LIN {X 0,Y 566.195,Z 59.453,A -85,B 0,C 180,E1 -2656.049,E2 -2656.049} C_VEL
LIN {X 0,Y 566.205,Z 59.459,A -85,B 0,C 180,E1 -2659.214,E2 -2659.214} C_VEL
LIN {X 0,Y 566.19,Z 59.456,A -85,B 0,C 180,E1 -2661.637,E2 -2661.637} C_VEL
LIN {X 0,Y 566.175,Z 59.454,A -85,B 0,C 180,E1 -2664.308,E2 -2664.308} C_VEL
LIN {X 0,Y 566.22,Z 59.453,A -85,B 0,C 180,E1 -2666.897,E2 -2666.897} C_VEL
LIN {X 0,Y 566.182,Z 59.457,A -85,B 0,C 180,E1 -2669.407,E2 -2669.407} C_VEL
LIN {X 0,Y 566.213,Z 59.448,A -85,B 0,C 180,E1 -2671.857,E2 -2671.857} C_VEL
LIN {X 0,Y 566.214,Z 59.449,A -85,B 0,C 180,E1 -2674.251,E2 -2674.251} C_VEL
LIN {X 0,Y 566.192,Z 59.462,A -85,B 0,C 180,E1 -2676.714,E2 -2676.714} C_VEL
LIN {X 0,Y 566.214,Z 59.447,A -85,B 0,C 180,E1 -2679.663,E2 -2679.663} C_VEL
LIN {X 0,Y 566.201,Z 59.457,A -85,B 0,C 180,E1 -2682.668,E2 -2682.668} C_VEL
LIN {X 0,Y 566.235,Z 59.447,A -85,B 0,C 180,E1 -2685.626,E2 -2685.626} C_VEL
LIN {X 0,Y 566.235,Z 59.447,A -85,B 0,C 180,E1 -2688.675,E2 -2688.675} C_VEL
LIN {X 0,Y 566.229,Z 59.444,A -85,B 0,C 180,E1 -2691.434,E2 -2691.434} C_VEL
LIN {X 0,Y 566.259,Z 59.451,A -85,B 0,C 180,E1 -2694.301,E2 -2694.301} C_VEL
LIN {X 0,Y 566.284,Z 59.447,A -85,B 0,C 180,E1 -2697.866,E2 -2697.866} C_VEL
LIN {X 0,Y 566.301,Z 59.435,A -85,B 0,C 180,E1 -2700.711,E2 -2700.711} C_VEL
LIN {X 0,Y 566.27,Z 59.442,A -85,B 0,C 180,E1 -2702.845,E2 -2702.845} C_VEL
LIN {X 0,Y 566.258,Z 59.453,A -85,B 0,C 180,E1 -2705.698,E2 -2705.698} C_VEL
LIN {X 0,Y 566.228,Z 59.445,A -85,B 0,C 180,E1 -2708.565,E2 -2708.565} C_VEL
LIN {X 0,Y 566.241,Z 59.45,A -85,B 0,C 180,E1 -2711.454,E2 -2711.454} C_VEL
LIN {X 0,Y 566.233,Z 59.447,A -85,B 0,C 180,E1 -2714.506,E2 -2714.506} C_VEL
LIN {X 0,Y 566.199,Z 59.459,A -85,B 0,C 180,E1 -2717.331,E2 -2717.331} C_VEL
LIN {X 0,Y 566.212,Z 59.447,A -85,B 0,C 180,E1 -2720.337,E2 -2720.337} C_VEL
LIN {X 0,Y 566.188,Z 59.459,A -85,B 0,C 180,E1 -2723.403,E2 -2723.403} C_VEL
LIN {X 0,Y 566.212,Z 59.449,A -85,B 0,C 180,E1 -2725.749,E2 -2725.749} C_VEL
LIN {X 0,Y 566.205,Z 59.452,A -85,B 0,C 180,E1 -2727.48,E2 -2727.48} C_VEL
LIN {X 0,Y 565.532,Z 59.535,A -85,B 0,C 180,E1 -2728.074,E2 -2728.074} C_VEL
LIN {X 0,Y 562.666,Z 59.9,A -85,B 0,C 180,E1 -2729.037,E2 -2729.037} C_VEL
LIN {X 0,Y 560.251,Z 60.196,A -85,B 0,C 180,E1 -2729.813,E2 -2729.813} C_VEL
LIN {X 0,Y 559.223,Z 60.323,A -85,B 0,C 180,E1 -2730.411,E2 -2730.411} C_VEL
LIN {X 0,Y 559.143,Z 60.333,A -85,B 0,C 180,E1 -2730.614,E2 -2730.614} C_VEL
LIN {X 0,Y 559.163,Z 60.326,A -85,B 0,C 180,E1 -2733.574,E2 -2733.574} C_VEL
LIN {X 0,Y 559.167,Z 60.331,A -85,B 0,C 180,E1 -2736.448,E2 -2736.448} C_VEL
LIN {X 0,Y 559.175,Z 60.331,A -85,B 0,C 180,E1 -2738.933,E2 -2738.933} C_VEL
LIN {X 0,Y 559.184,Z 60.325,A -85,B 0,C 180,E1 -2741.768,E2 -2741.768} C_VEL
LIN {X 0,Y 559.136,Z 60.335,A -85,B 0,C 180,E1 -2744.739,E2 -2744.739} C_VEL
LIN {X 0,Y 559.158,Z 60.322,A -85,B 0,C 180,E1 -2747.256,E2 -2747.256} C_VEL
LIN {X 0,Y 559.182,Z 60.329,A -85,B 0,C 180,E1 -2750.135,E2 -2750.135} C_VEL
LIN {X 0,Y 559.144,Z 60.331,A -85,B 0,C 180,E1 -2752.892,E2 -2752.892} C_VEL
LIN {X 0,Y 559.154,Z 60.326,A -85,B 0,C 180,E1 -2755.556,E2 -2755.556} C_VEL
LIN {X 0,Y 559.167,Z 60.336,A -85,B 0,C 180,E1 -2758.137,E2 -2758.137} C_VEL
LIN {X 0,Y 559.14,Z 60.329,A -85,B 0,C 180,E1 -2760.646,E2 -2760.646} C_VEL
LIN {X 0,Y 559.168,Z 60.329,A -85,B 0,C 180,E1 -2763.172,E2 -2763.172} C_VEL
LIN {X 0,Y 559.154,Z 60.335,A -85,B 0,C 180,E1 -2765.495,E2 -2765.495} C_VEL
LIN {X 0,Y 559.169,Z 60.328,A -85,B 0,C 180,E1 -2768.624,E2 -2768.624} C_VEL
LIN {X 0,Y 559.166,Z 60.33,A -85,B 0,C 180,E1 -2770.926,E2 -2770.926} C_VEL
LIN {X 0,Y 559.165,Z 60.332,A -85,B 0,C 180,E1 -2773.948,E2 -2773.948} C_VEL
LIN {X 0,Y 559.17,Z 60.329,A -85,B 0,C 180,E1 -2776.184,E2 -2776.184} C_VEL
LIN {X 0,Y 559.193,Z 60.332,A -85,B 0,C 180,E1 -2779.134,E2 -2779.134} C_VEL
LIN {X 0,Y 559.203,Z 60.325,A -85,B 0,C 180,E1 -2782.054,E2 -2782.054} C_VEL
LIN {X 0,Y 559.253,Z 60.324,A -85,B 0,C 180,E1 -2784.953,E2 -2784.953} C_VEL
LIN {X 0,Y 559.254,Z 60.319,A -85,B 0,C 180,E1 -2787.839,E2 -2787.839} C_VEL
LIN {X 0,Y 559.27,Z 60.322,A -85,B 0,C 180,E1 -2790.72,E2 -2790.72} C_VEL
LIN {X 0,Y 559.235,Z 60.328,A -85,B 0,C 180,E1 -2792.881,E2 -2792.881} C_VEL
LIN {X 0,Y 559.235,Z 60.321,A -85,B 0,C 180,E1 -2795.77,E2 -2795.77} C_VEL
LIN {X 0,Y 559.189,Z 60.334,A -85,B 0,C 180,E1 -2798.674,E2 -2798.674} C_VEL
LIN {X 0,Y 559.202,Z 60.324,A -85,B 0,C 180,E1 -2801.6,E2 -2801.6} C_VEL
LIN {X 0,Y 559.197,Z 60.333,A -85,B 0,C 180,E1 -2804.596,E2 -2804.596} C_VEL
LIN {X 0,Y 559.157,Z 60.33,A -85,B 0,C 180,E1 -2807.557,E2 -2807.557} C_VEL
LIN {X 0,Y 559.17,Z 60.331,A -85,B 0,C 180,E1 -2809.837,E2 -2809.837} C_VEL
LIN {X 0,Y 559.139,Z 60.34,A -85,B 0,C 180,E1 -2812.153,E2 -2812.153} C_VEL
LIN {X 0,Y 559.176,Z 60.327,A -85,B 0,C 180,E1 -2815.187,E2 -2815.187} C_VEL
LIN {X 0,Y 559.189,Z 60.329,A -85,B 0,C 180,E1 -2817.712,E2 -2817.712} C_VEL
LIN {X 0,Y 559.16,Z 60.329,A -85,B 0,C 180,E1 -2821.019,E2 -2821.019} C_VEL
LIN {X 0,Y 559.165,Z 60.33,A -85,B 0,C 180,E1 -2823.95,E2 -2823.95} C_VEL
LIN {X 0,Y 559.166,Z 60.329,A -85,B 0,C 180,E1 -2826.449,E2 -2826.449} C_VEL
LIN {X 0,Y 559.175,Z 60.327,A -85,B 0,C 180,E1 -2828.934,E2 -2828.934} C_VEL
LIN {X 0,Y 559.166,Z 60.327,A -85,B 0,C 180,E1 -2831.77,E2 -2831.77} C_VEL
LIN {X 0,Y 559.136,Z 60.33,A -85,B 0,C 180,E1 -2834.739,E2 -2834.739} C_VEL
LIN {X 0,Y 559.171,Z 60.329,A -85,B 0,C 180,E1 -2837.863,E2 -2837.863} C_VEL
LIN {X 0,Y 559.183,Z 60.325,A -85,B 0,C 180,E1 -2840.135,E2 -2840.135} C_VEL
LIN {X 0,Y 559.144,Z 60.335,A -85,B 0,C 180,E1 -2842.892,E2 -2842.892} C_VEL
LIN {X 0,Y 559.155,Z 60.33,A -85,B 0,C 180,E1 -2845.556,E2 -2845.556} C_VEL
LIN {X 0,Y 559.167,Z 60.328,A -85,B 0,C 180,E1 -2848.138,E2 -2848.138} C_VEL
LIN {X 0,Y 559.141,Z 60.335,A -85,B 0,C 180,E1 -2850.647,E2 -2850.647} C_VEL
LIN {X 0,Y 559.169,Z 60.331,A -85,B 0,C 180,E1 -2853.173,E2 -2853.173} C_VEL
LIN {X 0,Y 559.155,Z 60.33,A -85,B 0,C 180,E1 -2855.495,E2 -2855.495} C_VEL
LIN {X 0,Y 559.17,Z 60.335,A -85,B 0,C 180,E1 -2858.624,E2 -2858.624} C_VEL
LIN {X 0,Y 559.167,Z 60.329,A -85,B 0,C 180,E1 -2860.927,E2 -2860.927} C_VEL
LIN {X 0,Y 559.166,Z 60.328,A -85,B 0,C 180,E1 -2863.948,E2 -2863.948} C_VEL
LIN {X 0,Y 559.171,Z 60.332,A -85,B 0,C 180,E1 -2866.185,E2 -2866.185} C_VEL
LIN {X 0,Y 559.194,Z 60.32,A -85,B 0,C 180,E1 -2869.134,E2 -2869.134} C_VEL
LIN {X 0,Y 559.204,Z 60.325,A -85,B 0,C 180,E1 -2872.054,E2 -2872.054} C_VEL
LIN {X 0,Y 559.252,Z 60.318,A -85,B 0,C 180,E1 -2874.954,E2 -2874.954} C_VEL
LIN {X 0,Y 559.253,Z 60.321,A -85,B 0,C 180,E1 -2877.84,E2 -2877.84} C_VEL
LIN {X 0,Y 559.272,Z 60.311,A -85,B 0,C 180,E1 -2880.72,E2 -2880.72} C_VEL
LIN {X 0,Y 559.237,Z 60.318,A -85,B 0,C 180,E1 -2882.882,E2 -2882.882} C_VEL
LIN {X 0,Y 559.229,Z 60.328,A -85,B 0,C 180,E1 -2885.771,E2 -2885.771} C_VEL
LIN {X 0,Y 559.187,Z 60.321,A -85,B 0,C 180,E1 -2888.675,E2 -2888.675} C_VEL
LIN {X 0,Y 559.206,Z 60.327,A -85,B 0,C 180,E1 -2891.601,E2 -2891.601} C_VEL
LIN {X 0,Y 559.201,Z 60.323,A -85,B 0,C 180,E1 -2894.596,E2 -2894.596} C_VEL
LIN {X 0,Y 559.16,Z 60.331,A -85,B 0,C 180,E1 -2897.557,E2 -2897.557} C_VEL
LIN {X 0,Y 559.173,Z 60.327,A -85,B 0,C 180,E1 -2899.838,E2 -2899.838} C_VEL
LIN {X 0,Y 559.143,Z 60.33,A -85,B 0,C 180,E1 -2902.153,E2 -2902.153} C_VEL
LIN {X 0,Y 559.181,Z 60.333,A -85,B 0,C 180,E1 -2905.187,E2 -2905.187} C_VEL
LIN {X 0,Y 559.158,Z 60.328,A -85,B 0,C 180,E1 -2907.714,E2 -2907.714} C_VEL
LIN {X 0,Y 559.154,Z 60.329,A -85,B 0,C 180,E1 -2910.183,E2 -2910.183} C_VEL
LIN {X 0,Y 559.157,Z 60.334,A -85,B 0,C 180,E1 -2912.716,E2 -2912.716} C_VEL
LIN {X 0,Y 559.138,Z 60.334,A -85,B 0,C 180,E1 -2915.324,E2 -2915.324} C_VEL
LIN {X 0,Y 559.136,Z 60.332,A -85,B 0,C 180,E1 -2918.018,E2 -2918.018} C_VEL
LIN {X 0,Y 559.157,Z 60.337,A -85,B 0,C 180,E1 -2920.813,E2 -2920.813} C_VEL
LIN {X 0,Y 559.139,Z 60.331,A -85,B 0,C 180,E1 -2923.735,E2 -2923.735} C_VEL
LIN {X 0,Y 559.147,Z 60.335,A -85,B 0,C 180,E1 -2926.804,E2 -2926.804} C_VEL
LIN {X 0,Y 559.157,Z 60.326,A -85,B 0,C 180,E1 -2929.188,E2 -2929.188} C_VEL
LIN {X 0,Y 559.133,Z 60.336,A -85,B 0,C 180,E1 -2931.983,E2 -2931.983} C_VEL
LIN {X 0,Y 559.15,Z 60.331,A -85,B 0,C 180,E1 -2934.785,E2 -2934.785} C_VEL
LIN {X 0,Y 559.158,Z 60.329,A -85,B 0,C 180,E1 -2937.365,E2 -2937.365} C_VEL
LIN {X 0,Y 559.151,Z 60.337,A -85,B 0,C 180,E1 -2940.143,E2 -2940.143} C_VEL
LIN {X 0,Y 559.172,Z 60.331,A -85,B 0,C 180,E1 -2943.098,E2 -2943.098} C_VEL
LIN {X 0,Y 559.214,Z 60.39,A -85,B 0,C 180,E1 -2944.806,E2 -2944.806} C_VEL
LIN {X 0,Y 559.874,Z 64.838,A -85,B 0,C 180,E1 -2945.726,E2 -2945.726} C_VEL
LIN {X 0,Y 559.622,Z 80.36,A -85,B 0,C 180,E1 -2948.642,E2 -2948.642} C_VEL
LIN {X 0,Y 559.461,Z 94.988,A -85,B 0,C 180,E1 -2951.317,E2 -2951.317} C_VEL
LIN {X 0,Y 559.335,Z 110.651,A -85,B 0,C 180,E1 -2954.14,E2 -2954.14} C_VEL
LIN {X 0,Y 559.223,Z 120.021,A -85,B 0,C 180,E1 -2955.791,E2 -2955.791} C_VEL
LIN {X 0,Y 559.578,Z 122.477,A -85,B 0,C 180,E1 -2955.87,E2 -2955.87} C_VEL
LIN {X 0,Y 560.268,Z 127.87,A -85,B 0,C 180,E1 -2955.957,E2 -2955.957} C_VEL
LIN {X 0,Y 560.043,Z 224.999,A -85,B 0,C 180,E1 -2957.222,E2 -2957.222} C_VEL
LIN {X 0,Y 559.964,Z 235.772,A -85,B 0,C 180,E1 -2957.45,E2 -2957.45} C_VEL
LIN {X 0,Y 559.887,Z 244.879,A -85,B 0,C 180,E1 -2957.725,E2 -2957.725} C_VEL
LIN {X 0,Y 559.753,Z 254.245,A -85,B 0,C 180,E1 -2958.09,E2 -2958.09} C_VEL
LIN {X 0,Y 559.646,Z 263.579,A -85,B 0,C 180,E1 -2958.547,E2 -2958.547} C_VEL
LIN {X 0,Y 559.486,Z 273.383,A -85,B 0,C 180,E1 -2959.139,E2 -2959.139} C_VEL
LIN {X 0,Y 559.384,Z 282.116,A -85,B 0,C 180,E1 -2959.778,E2 -2959.778} C_VEL
LIN {X 0,Y 559.243,Z 289.512,A -85,B 0,C 180,E1 -2960.415,E2 -2960.415} C_VEL
LIN {X 0,Y 559.138,Z 296.709,A -85,B 0,C 180,E1 -2961.143,E2 -2961.143} C_VEL
LIN {X 0,Y 559.049,Z 302.886,A -85,B 0,C 180,E1 -2961.87,E2 -2961.87} C_VEL
LIN {X 0,Y 558.974,Z 309.395,A -85,B 0,C 180,E1 -2962.777,E2 -2962.777} C_VEL
LIN {X 0,Y 558.894,Z 313.874,A -85,B 0,C 180,E1 -2963.502,E2 -2963.502} C_VEL
LIN {X 0,Y 558.868,Z 319.334,A -85,B 0,C 180,E1 -2964.588,E2 -2964.588} C_VEL
LIN {X 0,Y 558.868,Z 323.629,A -85,B 0,C 180,E1 -2965.673,E2 -2965.673} C_VEL
LIN {X 0,Y 558.836,Z 325.974,A -85,B 0,C 180,E1 -2966.395,E2 -2966.395} C_VEL
LIN {X 0,Y 558.799,Z 327.762,A -85,B 0,C 180,E1 -2967.116,E2 -2967.116} C_VEL
LIN {X 0,Y 558.745,Z 330.188,A -85,B 0,C 180,E1 -2968.558,E2 -2968.558} C_VEL
LIN {X 0,Y 558.741,Z 330.772,A -85,B 0,C 180,E1 -2969.279,E2 -2969.279} C_VEL
LIN {X 0,Y 558.741,Z 330.772,A -85,B 0,C 180,E1 -2970.721,E2 -2970.721} C_VEL
LIN {X 0,Y 558.745,Z 330.188,A -85,B 0,C 180,E1 -2971.442,E2 -2971.442} C_VEL
LIN {X 0,Y 558.799,Z 327.762,A -85,B 0,C 180,E1 -2972.884,E2 -2972.884} C_VEL
LIN {X 0,Y 558.844,Z 324.837,A -85,B 0,C 180,E1 -2973.966,E2 -2973.966} C_VEL
LIN {X 0,Y 558.797,Z 320.878,A -85,B 0,C 180,E1 -2975.051,E2 -2975.051} C_VEL
LIN {X 0,Y 558.91,Z 315.779,A -85,B 0,C 180,E1 -2976.136,E2 -2976.136} C_VEL
LIN {X 0,Y 558.934,Z 310.66,A -85,B 0,C 180,E1 -2977.024,E2 -2977.024} C_VEL
LIN {X 0,Y 559.052,Z 304.256,A -85,B 0,C 180,E1 -2977.949,E2 -2977.949} C_VEL
LIN {X 0,Y 559.104,Z 298.33,A -85,B 0,C 180,E1 -2978.676,E2 -2978.676} C_VEL
LIN {X 0,Y 559.228,Z 291.427,A -85,B 0,C 180,E1 -2979.403,E2 -2979.403} C_VEL
LIN {X 0,Y 559.335,Z 283.25,A -85,B 0,C 180,E1 -2980.132,E2 -2980.132} C_VEL
LIN {X 0,Y 559.461,Z 274.735,A -85,B 0,C 180,E1 -2980.77,E2 -2980.77} C_VEL
LIN {X 0,Y 559.613,Z 265.677,A -85,B 0,C 180,E1 -2981.336,E2 -2981.336} C_VEL
LIN {X 0,Y 559.75,Z 256.559,A -85,B 0,C 180,E1 -2981.805,E2 -2981.805} C_VEL
LIN {X 0,Y 559.829,Z 247.457,A -85,B 0,C 180,E1 -2982.184,E2 -2982.184} C_VEL
LIN {X 0,Y 559.948,Z 237.521,A -85,B 0,C 180,E1 -2982.504,E2 -2982.504} C_VEL
LIN {X 0,Y 560.025,Z 227.662,A -85,B 0,C 180,E1 -2982.732,E2 -2982.732} C_VEL
LIN {X 0,Y 560.141,Z 203.051,A -85,B 0,C 180,E1 -2983.075,E2 -2983.075} C_VEL
LIN {X 0,Y 560.204,Z 126.078,A -85,B 0,C 180,E1 -2984.068,E2 -2984.068} C_VEL
LIN {X 0,Y 559.255,Z 120.352,A -85,B 0,C 180,E1 -2984.185,E2 -2984.185} C_VEL
LIN {X 0,Y 559.19,Z 118.972,A -85,B 0,C 180,E1 -2984.372,E2 -2984.372} C_VEL
LIN {X 0,Y 559.322,Z 105.432,A -85,B 0,C 180,E1 -2986.798,E2 -2986.798} C_VEL
LIN {X 0,Y 559.555,Z 89.886,A -85,B 0,C 180,E1 -2989.609,E2 -2989.609} C_VEL
LIN {X 0,Y 559.737,Z 73.174,A -85,B 0,C 180,E1 -2992.712,E2 -2992.712} C_VEL
LIN {X 0,Y 559.796,Z 63.816,A -85,B 0,C 180,E1 -2994.475,E2 -2994.475} C_VEL
LIN {X 0,Y 559.204,Z 60.36,A -85,B 0,C 180,E1 -2995.191,E2 -2995.191} C_VEL
LIN {X 0,Y 559.184,Z 60.332,A -85,B 0,C 180,E1 -2997.712,E2 -2997.712} C_VEL
LIN {X 0,Y 559.157,Z 60.336,A -85,B 0,C 180,E1 -3000.182,E2 -3000.182} C_VEL
LIN {X 0,Y 559.159,Z 60.329,A -85,B 0,C 180,E1 -3002.715,E2 -3002.715} C_VEL
LIN {X 0,Y 559.147,Z 60.333,A -85,B 0,C 180,E1 -3005.323,E2 -3005.323} C_VEL
LIN {X 0,Y 559.133,Z 60.336,A -85,B 0,C 180,E1 -3008.017,E2 -3008.017} C_VEL
LIN {X 0,Y 559.157,Z 60.326,A -85,B 0,C 180,E1 -3010.812,E2 -3010.812} C_VEL
LIN {X 0,Y 559.139,Z 60.336,A -85,B 0,C 180,E1 -3013.734,E2 -3013.734} C_VEL
LIN {X 0,Y 559.146,Z 60.332,A -85,B 0,C 180,E1 -3016.803,E2 -3016.803} C_VEL
LIN {X 0,Y 559.157,Z 60.337,A -85,B 0,C 180,E1 -3019.187,E2 -3019.187} C_VEL
LIN {X 0,Y 559.136,Z 60.332,A -85,B 0,C 180,E1 -3021.982,E2 -3021.982} C_VEL
LIN {X 0,Y 559.143,Z 60.334,A -85,B 0,C 180,E1 -3024.785,E2 -3024.785} C_VEL
LIN {X 0,Y 559.156,Z 60.333,A -85,B 0,C 180,E1 -3027.364,E2 -3027.364} C_VEL
LIN {X 0,Y 559.149,Z 60.33,A -85,B 0,C 180,E1 -3030.142,E2 -3030.142} C_VEL
LIN {X 0,Y 559.17,Z 60.329,A -85,B 0,C 180,E1 -3033.097,E2 -3033.097} C_VEL
LIN {X 0,Y 559.158,Z 60.329,A -85,B 0,C 180,E1 -3035.495,E2 -3035.495} C_VEL
LIN {X 0,Y 559.173,Z 60.335,A -85,B 0,C 180,E1 -3038.624,E2 -3038.624} C_VEL
LIN {X 0,Y 559.167,Z 60.326,A -85,B 0,C 180,E1 -3040.926,E2 -3040.926} C_VEL
LIN {X 0,Y 559.167,Z 60.328,A -85,B 0,C 180,E1 -3043.948,E2 -3043.948} C_VEL
LIN {X 0,Y 559.173,Z 60.332,A -85,B 0,C 180,E1 -3046.184,E2 -3046.184} C_VEL
LIN {X 0,Y 559.196,Z 60.32,A -85,B 0,C 180,E1 -3049.133,E2 -3049.133} C_VEL
LIN {X 0,Y 559.204,Z 60.325,A -85,B 0,C 180,E1 -3052.053,E2 -3052.053} C_VEL
LIN {X 0,Y 559.252,Z 60.317,A -85,B 0,C 180,E1 -3054.953,E2 -3054.953} C_VEL
LIN {X 0,Y 559.255,Z 60.322,A -85,B 0,C 180,E1 -3057.839,E2 -3057.839} C_VEL
LIN {X 0,Y 559.272,Z 60.31,A -85,B 0,C 180,E1 -3060.72,E2 -3060.72} C_VEL
LIN {X 0,Y 559.237,Z 60.318,A -85,B 0,C 180,E1 -3062.881,E2 -3062.881} C_VEL
LIN {X 0,Y 559.228,Z 60.329,A -85,B 0,C 180,E1 -3065.77,E2 -3065.77} C_VEL
LIN {X 0,Y 559.187,Z 60.321,A -85,B 0,C 180,E1 -3068.674,E2 -3068.674} C_VEL
LIN {X 0,Y 559.205,Z 60.329,A -85,B 0,C 180,E1 -3071.6,E2 -3071.6} C_VEL
LIN {X 0,Y 559.199,Z 60.324,A -85,B 0,C 180,E1 -3074.595,E2 -3074.595} C_VEL
LIN {X 0,Y 559.158,Z 60.331,A -85,B 0,C 180,E1 -3077.556,E2 -3077.556} C_VEL
LIN {X 0,Y 559.171,Z 60.326,A -85,B 0,C 180,E1 -3079.837,E2 -3079.837} C_VEL
LIN {X 0,Y 559.14,Z 60.331,A -85,B 0,C 180,E1 -3082.152,E2 -3082.152} C_VEL
LIN {X 0,Y 559.177,Z 60.333,A -85,B 0,C 180,E1 -3085.187,E2 -3085.187} C_VEL
LIN {X 0,Y 559.187,Z 60.323,A -85,B 0,C 180,E1 -3087.711,E2 -3087.711} C_VEL
LIN {X 0,Y 559.143,Z 60.333,A -85,B 0,C 180,E1 -3090.614,E2 -3090.614} C_VEL
LIN {X 0,Y 558.484,Z 60.421,A -85,B 0,C 180,E1 -3091.216,E2 -3091.216} C_VEL
LIN {X 0,Y 555.622,Z 60.774,A -85,B 0,C 180,E1 -3092.192,E2 -3092.192} C_VEL
LIN {X 0,Y 553.209,Z 61.075,A -85,B 0,C 180,E1 -3092.977,E2 -3092.977} C_VEL
LIN {X 0,Y 552.188,Z 61.195,A -85,B 0,C 180,E1 -3093.584,E2 -3093.584} C_VEL
LIN {X 0,Y 552.113,Z 61.204,A -85,B 0,C 180,E1 -3093.789,E2 -3093.789} C_VEL
LIN {X 0,Y 552.11,Z 61.215,A -85,B 0,C 180,E1 -3096.746,E2 -3096.746} C_VEL
LIN {X 0,Y 552.132,Z 61.203,A -85,B 0,C 180,E1 -3099.526,E2 -3099.526} C_VEL
LIN {X 0,Y 552.127,Z 61.211,A -85,B 0,C 180,E1 -3102.425,E2 -3102.425} C_VEL
LIN {X 0,Y 552.094,Z 61.207,A -85,B 0,C 180,E1 -3105.562,E2 -3105.562} C_VEL
LIN {X 0,Y 552.137,Z 61.204,A -85,B 0,C 180,E1 -3108.676,E2 -3108.676} C_VEL
LIN {X 0,Y 552.117,Z 61.206,A -85,B 0,C 180,E1 -3111.411,E2 -3111.411} C_VEL
LIN {X 0,Y 552.111,Z 61.211,A -85,B 0,C 180,E1 -3114.158,E2 -3114.158} C_VEL
LIN {X 0,Y 552.12,Z 61.206,A -85,B 0,C 180,E1 -3116.815,E2 -3116.815} C_VEL
LIN {X 0,Y 552.104,Z 61.209,A -85,B 0,C 180,E1 -3119.391,E2 -3119.391} C_VEL
LIN {X 0,Y 552.123,Z 61.211,A -85,B 0,C 180,E1 -3121.903,E2 -3121.903} C_VEL
LIN {X 0,Y 552.152,Z 61.203,A -85,B 0,C 180,E1 -3124.649,E2 -3124.649} C_VEL
LIN {X 0,Y 552.093,Z 61.216,A -85,B 0,C 180,E1 -3127.549,E2 -3127.549} C_VEL
LIN {X 0,Y 552.153,Z 61.203,A -85,B 0,C 180,E1 -3130.674,E2 -3130.674} C_VEL
LIN {X 0,Y 552.115,Z 61.214,A -85,B 0,C 180,E1 -3133.737,E2 -3133.737} C_VEL
LIN {X 0,Y 552.133,Z 61.207,A -85,B 0,C 180,E1 -3136.004,E2 -3136.004} C_VEL
LIN {X 0,Y 552.16,Z 61.206,A -85,B 0,C 180,E1 -3138.993,E2 -3138.993} C_VEL
LIN {X 0,Y 552.157,Z 61.203,A -85,B 0,C 180,E1 -3141.952,E2 -3141.952} C_VEL
LIN {X 0,Y 552.229,Z 61.199,A -85,B 0,C 180,E1 -3144.889,E2 -3144.889} C_VEL
LIN {X 0,Y 552.225,Z 61.195,A -85,B 0,C 180,E1 -3147.812,E2 -3147.812} C_VEL
LIN {X 0,Y 552.24,Z 61.198,A -85,B 0,C 180,E1 -3150.729,E2 -3150.729} C_VEL
LIN {X 0,Y 552.202,Z 61.204,A -85,B 0,C 180,E1 -3152.918,E2 -3152.918} C_VEL
LIN {X 0,Y 552.205,Z 61.196,A -85,B 0,C 180,E1 -3155.844,E2 -3155.844} C_VEL
LIN {X 0,Y 552.16,Z 61.21,A -85,B 0,C 180,E1 -3158.786,E2 -3158.786} C_VEL
LIN {X 0,Y 552.16,Z 61.202,A -85,B 0,C 180,E1 -3161.751,E2 -3161.751} C_VEL
LIN {X 0,Y 552.134,Z 61.211,A -85,B 0,C 180,E1 -3164.748,E2 -3164.748} C_VEL
LIN {X 0,Y 552.108,Z 61.209,A -85,B 0,C 180,E1 -3167.788,E2 -3167.788} C_VEL
LIN {X 0,Y 552.128,Z 61.211,A -85,B 0,C 180,E1 -3170.101,E2 -3170.101} C_VEL
LIN {X 0,Y 552.093,Z 61.216,A -85,B 0,C 180,E1 -3172.451,E2 -3172.451} C_VEL
LIN {X 0,Y 552.152,Z 61.203,A -85,B 0,C 180,E1 -3175.351,E2 -3175.351} C_VEL
LIN {X 0,Y 552.123,Z 61.211,A -85,B 0,C 180,E1 -3178.097,E2 -3178.097} C_VEL
LIN {X 0,Y 552.104,Z 61.209,A -85,B 0,C 180,E1 -3180.609,E2 -3180.609} C_VEL
LIN {X 0,Y 552.12,Z 61.206,A -85,B 0,C 180,E1 -3183.185,E2 -3183.185} C_VEL
LIN {X 0,Y 552.111,Z 61.211,A -85,B 0,C 180,E1 -3185.842,E2 -3185.842} C_VEL
LIN {X 0,Y 552.123,Z 61.207,A -85,B 0,C 180,E1 -3189.062,E2 -3189.062} C_VEL
LIN {X 0,Y 552.127,Z 61.206,A -85,B 0,C 180,E1 -3191.445,E2 -3191.445} C_VEL
LIN {X 0,Y 552.092,Z 61.207,A -85,B 0,C 180,E1 -3194.532,E2 -3194.532} C_VEL
LIN {X 0,Y 552.128,Z 61.21,A -85,B 0,C 180,E1 -3197.585,E2 -3197.585} C_VEL
LIN {X 0,Y 552.131,Z 61.203,A -85,B 0,C 180,E1 -3200.474,E2 -3200.474} C_VEL
LIN {X 0,Y 552.112,Z 61.214,A -85,B 0,C 180,E1 -3203.316,E2 -3203.316} C_VEL
LIN {X 0,Y 552.13,Z 61.202,A -85,B 0,C 180,E1 -3205.94,E2 -3205.94} C_VEL
LIN {X 0,Y 552.116,Z 61.208,A -85,B 0,C 180,E1 -3208.541,E2 -3208.541} C_VEL
LIN {X 0,Y 552.122,Z 61.205,A -85,B 0,C 180,E1 -3211.438,E2 -3211.438} C_VEL
LIN {X 0,Y 552.128,Z 61.204,A -85,B 0,C 180,E1 -3214.356,E2 -3214.356} C_VEL
LIN {X 0,Y 552.109,Z 61.216,A -85,B 0,C 180,E1 -3216.759,E2 -3216.759} C_VEL
LIN {X 0,Y 552.119,Z 61.206,A -85,B 0,C 180,E1 -3219.12,E2 -3219.12} C_VEL
LIN {X 0,Y 552.124,Z 61.201,A -85,B 0,C 180,E1 -3221.445,E2 -3221.445} C_VEL
LIN {X 0,Y 552.116,Z 61.205,A -85,B 0,C 180,E1 -3223.738,E2 -3223.738} C_VEL
LIN {X 0,Y 552.135,Z 61.206,A -85,B 0,C 180,E1 -3226.005,E2 -3226.005} C_VEL
LIN {X 0,Y 552.162,Z 61.197,A -85,B 0,C 180,E1 -3228.994,E2 -3228.994} C_VEL
LIN {X 0,Y 552.157,Z 61.2,A -85,B 0,C 180,E1 -3231.952,E2 -3231.952} C_VEL
LIN {X 0,Y 552.227,Z 61.193,A -85,B 0,C 180,E1 -3234.889,E2 -3234.889} C_VEL
LIN {X 0,Y 552.225,Z 61.196,A -85,B 0,C 180,E1 -3237.812,E2 -3237.812} C_VEL
LIN {X 0,Y 552.242,Z 61.186,A -85,B 0,C 180,E1 -3240.73,E2 -3240.73} C_VEL
LIN {X 0,Y 552.203,Z 61.194,A -85,B 0,C 180,E1 -3242.919,E2 -3242.919} C_VEL
LIN {X 0,Y 552.2,Z 61.204,A -85,B 0,C 180,E1 -3245.844,E2 -3245.844} C_VEL
LIN {X 0,Y 552.158,Z 61.196,A -85,B 0,C 180,E1 -3248.786,E2 -3248.786} C_VEL
LIN {X 0,Y 552.163,Z 61.207,A -85,B 0,C 180,E1 -3251.751,E2 -3251.751} C_VEL
LIN {X 0,Y 552.137,Z 61.203,A -85,B 0,C 180,E1 -3254.749,E2 -3254.749} C_VEL
LIN {X 0,Y 552.11,Z 61.205,A -85,B 0,C 180,E1 -3257.789,E2 -3257.789} C_VEL
LIN {X 0,Y 552.132,Z 61.202,A -85,B 0,C 180,E1 -3260.102,E2 -3260.102} C_VEL
LIN {X 0,Y 552.097,Z 61.208,A -85,B 0,C 180,E1 -3262.451,E2 -3262.451} C_VEL
LIN {X 0,Y 552.157,Z 61.204,A -85,B 0,C 180,E1 -3265.351,E2 -3265.351} C_VEL
LIN {X 0,Y 552.11,Z 61.204,A -85,B 0,C 180,E1 -3268.099,E2 -3268.099} C_VEL
LIN {X 0,Y 552.104,Z 61.211,A -85,B 0,C 180,E1 -3270.61,E2 -3270.61} C_VEL
LIN {X 0,Y 552.116,Z 61.208,A -85,B 0,C 180,E1 -3273.186,E2 -3273.186} C_VEL
LIN {X 0,Y 552.09,Z 61.208,A -85,B 0,C 180,E1 -3275.844,E2 -3275.844} C_VEL
LIN {X 0,Y 552.127,Z 61.207,A -85,B 0,C 180,E1 -3279.062,E2 -3279.062} C_VEL
LIN {X 0,Y 552.122,Z 61.206,A -85,B 0,C 180,E1 -3281.446,E2 -3281.446} C_VEL
LIN {X 0,Y 552.09,Z 61.217,A -85,B 0,C 180,E1 -3284.531,E2 -3284.531} C_VEL
LIN {X 0,Y 552.131,Z 61.204,A -85,B 0,C 180,E1 -3287.585,E2 -3287.585} C_VEL
LIN {X 0,Y 552.131,Z 61.209,A -85,B 0,C 180,E1 -3290.473,E2 -3290.473} C_VEL
LIN {X 0,Y 552.113,Z 61.207,A -85,B 0,C 180,E1 -3293.317,E2 -3293.317} C_VEL
LIN {X 0,Y 552.133,Z 61.208,A -85,B 0,C 180,E1 -3295.94,E2 -3295.94} C_VEL
LIN {X 0,Y 552.122,Z 61.21,A -85,B 0,C 180,E1 -3298.541,E2 -3298.541} C_VEL
LIN {X 0,Y 552.127,Z 61.209,A -85,B 0,C 180,E1 -3301.438,E2 -3301.438} C_VEL
LIN {X 0,Y 552.136,Z 61.212,A -85,B 0,C 180,E1 -3304.356,E2 -3304.356} C_VEL
LIN {X 0,Y 552.208,Z 61.501,A -85,B 0,C 180,E1 -3304.732,E2 -3304.732} C_VEL
LIN {X 0,Y 552.933,Z 66.827,A -85,B 0,C 180,E1 -3305.801,E2 -3305.801} C_VEL
LIN {X 0,Y 552.656,Z 81.314,A -85,B 0,C 180,E1 -3308.555,E2 -3308.555} C_VEL
LIN {X 0,Y 552.457,Z 94.858,A -85,B 0,C 180,E1 -3311.071,E2 -3311.071} C_VEL
LIN {X 0,Y 552.324,Z 110.523,A -85,B 0,C 180,E1 -3313.933,E2 -3313.933} C_VEL
LIN {X 0,Y 552.154,Z 119.891,A -85,B 0,C 180,E1 -3315.611,E2 -3315.611} C_VEL
LIN {X 0,Y 553.008,Z 125.151,A -85,B 0,C 180,E1 -3315.736,E2 -3315.736} C_VEL
LIN {X 0,Y 553.361,Z 129.745,A -85,B 0,C 180,E1 -3315.805,E2 -3315.805} C_VEL
LIN {X 0,Y 553.136,Z 224.808,A -85,B 0,C 180,E1 -3317.06,E2 -3317.06} C_VEL
LIN {X 0,Y 553.048,Z 234.707,A -85,B 0,C 180,E1 -3317.268,E2 -3317.268} C_VEL
LIN {X 0,Y 552.931,Z 244.686,A -85,B 0,C 180,E1 -3317.568,E2 -3317.568} C_VEL
LIN {X 0,Y 552.802,Z 254.046,A -85,B 0,C 180,E1 -3317.938,E2 -3317.938} C_VEL
LIN {X 0,Y 552.643,Z 264.468,A -85,B 0,C 180,E1 -3318.462,E2 -3318.462} C_VEL
LIN {X 0,Y 552.489,Z 273.192,A -85,B 0,C 180,E1 -3319,E2 -3319} C_VEL
LIN {X 0,Y 552.342,Z 281.924,A -85,B 0,C 180,E1 -3319.646,E2 -3319.646} C_VEL
LIN {X 0,Y 552.204,Z 289.321,A -85,B 0,C 180,E1 -3320.292,E2 -3320.292} C_VEL
LIN {X 0,Y 552.099,Z 296.543,A -85,B 0,C 180,E1 -3321.029,E2 -3321.029} C_VEL
LIN {X 0,Y 552.012,Z 302.745,A -85,B 0,C 180,E1 -3321.765,E2 -3321.765} C_VEL
LIN {X 0,Y 551.904,Z 309.281,A -85,B 0,C 180,E1 -3322.684,E2 -3322.684} C_VEL
LIN {X 0,Y 551.805,Z 314.997,A -85,B 0,C 180,E1 -3323.651,E2 -3323.651} C_VEL
LIN {X 0,Y 551.802,Z 319.269,A -85,B 0,C 180,E1 -3324.519,E2 -3324.519} C_VEL
LIN {X 0,Y 551.765,Z 323.587,A -85,B 0,C 180,E1 -3325.617,E2 -3325.617} C_VEL
LIN {X 0,Y 551.75,Z 325.95,A -85,B 0,C 180,E1 -3326.348,E2 -3326.348} C_VEL
LIN {X 0,Y 551.723,Z 327.744,A -85,B 0,C 180,E1 -3327.079,E2 -3327.079} C_VEL
LIN {X 0,Y 551.645,Z 330.177,A -85,B 0,C 180,E1 -3328.54,E2 -3328.54} C_VEL
LIN {X 0,Y 551.641,Z 330.761,A -85,B 0,C 180,E1 -3329.27,E2 -3329.27} C_VEL
LIN {X 0,Y 551.641,Z 330.761,A -85,B 0,C 180,E1 -3330.73,E2 -3330.73} C_VEL
LIN {X 0,Y 551.645,Z 330.177,A -85,B 0,C 180,E1 -3331.46,E2 -3331.46} C_VEL
LIN {X 0,Y 551.723,Z 327.744,A -85,B 0,C 180,E1 -3332.921,E2 -3332.921} C_VEL
LIN {X 0,Y 551.764,Z 324.802,A -85,B 0,C 180,E1 -3334.017,E2 -3334.017} C_VEL
LIN {X 0,Y 551.723,Z 320.819,A -85,B 0,C 180,E1 -3335.116,E2 -3335.116} C_VEL
LIN {X 0,Y 551.837,Z 316.303,A -85,B 0,C 180,E1 -3336.098,E2 -3336.098} C_VEL
LIN {X 0,Y 551.886,Z 310.436,A -85,B 0,C 180,E1 -3337.132,E2 -3337.132} C_VEL
LIN {X 0,Y 551.984,Z 304.121,A -85,B 0,C 180,E1 -3338.051,E2 -3338.051} C_VEL
LIN {X 0,Y 552.055,Z 298.169,A -85,B 0,C 180,E1 -3338.787,E2 -3338.787} C_VEL
LIN {X 0,Y 552.172,Z 291.241,A -85,B 0,C 180,E1 -3339.524,E2 -3339.524} C_VEL
LIN {X 0,Y 552.333,Z 283.059,A -85,B 0,C 180,E1 -3340.261,E2 -3340.261} C_VEL
LIN {X 0,Y 552.462,Z 274.544,A -85,B 0,C 180,E1 -3340.908,E2 -3340.908} C_VEL
LIN {X 0,Y 552.624,Z 265.626,A -85,B 0,C 180,E1 -3341.473,E2 -3341.473} C_VEL
LIN {X 0,Y 552.789,Z 256.061,A -85,B 0,C 180,E1 -3341.97,E2 -3341.97} C_VEL
LIN {X 0,Y 552.892,Z 247.263,A -85,B 0,C 180,E1 -3342.34,E2 -3342.34} C_VEL
LIN {X 0,Y 553.004,Z 237.33,A -85,B 0,C 180,E1 -3342.664,E2 -3342.664} C_VEL
LIN {X 0,Y 553.096,Z 227.472,A -85,B 0,C 180,E1 -3342.895,E2 -3342.895} C_VEL
LIN {X 0,Y 553.222,Z 202.86,A -85,B 0,C 180,E1 -3343.242,E2 -3343.242} C_VEL
LIN {X 0,Y 553.263,Z 126.541,A -85,B 0,C 180,E1 -3344.239,E2 -3344.239} C_VEL
LIN {X 0,Y 552.178,Z 120.063,A -85,B 0,C 180,E1 -3344.376,E2 -3344.376} C_VEL
LIN {X 0,Y 552.204,Z 115.738,A -85,B 0,C 180,E1 -3345.124,E2 -3345.124} C_VEL
LIN {X 0,Y 552.442,Z 100.083,A -85,B 0,C 180,E1 -3347.969,E2 -3347.969} C_VEL
LIN {X 0,Y 552.591,Z 85.455,A -85,B 0,C 180,E1 -3350.667,E2 -3350.667} C_VEL
LIN {X 0,Y 552.895,Z 70.564,A -85,B 0,C 180,E1 -3353.487,E2 -3353.487} C_VEL
LIN {X 0,Y 552.781,Z 64.77,A -85,B 0,C 180,E1 -3354.606,E2 -3354.606} C_VEL
LIN {X 0,Y 552.163,Z 61.23,A -85,B 0,C 180,E1 -3355.363,E2 -3355.363} C_VEL
LIN {X 0,Y 552.123,Z 61.213,A -85,B 0,C 180,E1 -3358.097,E2 -3358.097} C_VEL
LIN {X 0,Y 552.106,Z 61.21,A -85,B 0,C 180,E1 -3360.609,E2 -3360.609} C_VEL
LIN {X 0,Y 552.118,Z 61.208,A -85,B 0,C 180,E1 -3363.186,E2 -3363.186} C_VEL
LIN {X 0,Y 552.102,Z 61.214,A -85,B 0,C 180,E1 -3365.842,E2 -3365.842} C_VEL
LIN {X 0,Y 552.122,Z 61.207,A -85,B 0,C 180,E1 -3369.061,E2 -3369.061} C_VEL
LIN {X 0,Y 552.123,Z 61.209,A -85,B 0,C 180,E1 -3371.446,E2 -3371.446} C_VEL
LIN {X 0,Y 552.09,Z 61.209,A -85,B 0,C 180,E1 -3374.531,E2 -3374.531} C_VEL
LIN {X 0,Y 552.131,Z 61.21,A -85,B 0,C 180,E1 -3377.584,E2 -3377.584} C_VEL
LIN {X 0,Y 552.135,Z 61.202,A -85,B 0,C 180,E1 -3380.473,E2 -3380.473} C_VEL
LIN {X 0,Y 552.108,Z 61.213,A -85,B 0,C 180,E1 -3383.317,E2 -3383.317} C_VEL
LIN {X 0,Y 552.131,Z 61.201,A -85,B 0,C 180,E1 -3385.939,E2 -3385.939} C_VEL
LIN {X 0,Y 552.12,Z 61.208,A -85,B 0,C 180,E1 -3388.54,E2 -3388.54} C_VEL
LIN {X 0,Y 552.125,Z 61.204,A -85,B 0,C 180,E1 -3391.438,E2 -3391.438} C_VEL
LIN {X 0,Y 552.131,Z 61.203,A -85,B 0,C 180,E1 -3394.355,E2 -3394.355} C_VEL
LIN {X 0,Y 552.111,Z 61.215,A -85,B 0,C 180,E1 -3396.758,E2 -3396.758} C_VEL
LIN {X 0,Y 552.121,Z 61.205,A -85,B 0,C 180,E1 -3399.119,E2 -3399.119} C_VEL
LIN {X 0,Y 552.123,Z 61.199,A -85,B 0,C 180,E1 -3401.444,E2 -3401.444} C_VEL
LIN {X 0,Y 552.117,Z 61.204,A -85,B 0,C 180,E1 -3403.737,E2 -3403.737} C_VEL
LIN {X 0,Y 552.136,Z 61.206,A -85,B 0,C 180,E1 -3406.004,E2 -3406.004} C_VEL
LIN {X 0,Y 552.163,Z 61.196,A -85,B 0,C 180,E1 -3408.993,E2 -3408.993} C_VEL
LIN {X 0,Y 552.158,Z 61.201,A -85,B 0,C 180,E1 -3411.951,E2 -3411.951} C_VEL
LIN {X 0,Y 552.227,Z 61.193,A -85,B 0,C 180,E1 -3414.889,E2 -3414.889} C_VEL
LIN {X 0,Y 552.226,Z 61.197,A -85,B 0,C 180,E1 -3417.812,E2 -3417.812} C_VEL
LIN {X 0,Y 552.242,Z 61.185,A -85,B 0,C 180,E1 -3420.729,E2 -3420.729} C_VEL
LIN {X 0,Y 552.203,Z 61.194,A -85,B 0,C 180,E1 -3422.918,E2 -3422.918} C_VEL
LIN {X 0,Y 552.199,Z 61.203,A -85,B 0,C 180,E1 -3425.843,E2 -3425.843} C_VEL
LIN {X 0,Y 552.157,Z 61.197,A -85,B 0,C 180,E1 -3428.785,E2 -3428.785} C_VEL
LIN {X 0,Y 552.162,Z 61.206,A -85,B 0,C 180,E1 -3431.75,E2 -3431.75} C_VEL
LIN {X 0,Y 552.136,Z 61.204,A -85,B 0,C 180,E1 -3434.748,E2 -3434.748} C_VEL
LIN {X 0,Y 552.109,Z 61.205,A -85,B 0,C 180,E1 -3437.788,E2 -3437.788} C_VEL
LIN {X 0,Y 552.13,Z 61.201,A -85,B 0,C 180,E1 -3440.101,E2 -3440.101} C_VEL
LIN {X 0,Y 552.094,Z 61.209,A -85,B 0,C 180,E1 -3442.45,E2 -3442.45} C_VEL
LIN {X 0,Y 552.154,Z 61.204,A -85,B 0,C 180,E1 -3445.35,E2 -3445.35} C_VEL
LIN {X 0,Y 552.121,Z 61.202,A -85,B 0,C 180,E1 -3448.097,E2 -3448.097} C_VEL
LIN {X 0,Y 552.106,Z 61.211,A -85,B 0,C 180,E1 -3450.61,E2 -3450.61} C_VEL
LIN {X 0,Y 552.121,Z 61.207,A -85,B 0,C 180,E1 -3453.185,E2 -3453.185} C_VEL
LIN {X 0,Y 552.113,Z 61.204,A -85,B 0,C 180,E1 -3453.789,E2 -3453.789} C_VEL
LIN {X 0,Y 551.478,Z 61.287,A -85,B 0,C 180,E1 -3454.398,E2 -3454.398} C_VEL
LIN {X 0,Y 548.657,Z 61.645,A -85,B 0,C 180,E1 -3455.386,E2 -3455.386} C_VEL
LIN {X 0,Y 546.236,Z 61.95,A -85,B 0,C 180,E1 -3456.182,E2 -3456.182} C_VEL
LIN {X 0,Y 545.166,Z 62.081,A -85,B 0,C 180,E1 -3456.796,E2 -3456.796} C_VEL
LIN {X 0,Y 545.063,Z 62.09,A -85,B 0,C 180,E1 -3457.004,E2 -3457.004} C_VEL
LIN {X 0,Y 545.072,Z 62.085,A -85,B 0,C 180,E1 -3460.141,E2 -3460.141} C_VEL
LIN {X 0,Y 545.075,Z 62.085,A -85,B 0,C 180,E1 -3463.106,E2 -3463.106} C_VEL
LIN {X 0,Y 545.053,Z 62.089,A -85,B 0,C 180,E1 -3466.225,E2 -3466.225} C_VEL
LIN {X 0,Y 545.094,Z 62.078,A -85,B 0,C 180,E1 -3468.887,E2 -3468.887} C_VEL
LIN {X 0,Y 545.051,Z 62.089,A -85,B 0,C 180,E1 -3471.763,E2 -3471.763} C_VEL
LIN {X 0,Y 545.063,Z 62.082,A -85,B 0,C 180,E1 -3474.534,E2 -3474.534} C_VEL
LIN {X 0,Y 545.078,Z 62.082,A -85,B 0,C 180,E1 -3477.212,E2 -3477.212} C_VEL
LIN {X 0,Y 545.063,Z 62.091,A -85,B 0,C 180,E1 -3479.811,E2 -3479.811} C_VEL
LIN {X 0,Y 545.091,Z 62.085,A -85,B 0,C 180,E1 -3482.344,E2 -3482.344} C_VEL
LIN {X 0,Y 545.114,Z 62.079,A -85,B 0,C 180,E1 -3484.82,E2 -3484.82} C_VEL
LIN {X 0,Y 545.041,Z 62.091,A -85,B 0,C 180,E1 -3487.243,E2 -3487.243} C_VEL
LIN {X 0,Y 545.117,Z 62.08,A -85,B 0,C 180,E1 -3490.415,E2 -3490.415} C_VEL
LIN {X 0,Y 545.072,Z 62.093,A -85,B 0,C 180,E1 -3493.521,E2 -3493.521} C_VEL
LIN {X 0,Y 545.092,Z 62.086,A -85,B 0,C 180,E1 -3495.82,E2 -3495.82} C_VEL
LIN {X 0,Y 545.115,Z 62.082,A -85,B 0,C 180,E1 -3498.849,E2 -3498.849} C_VEL
LIN {X 0,Y 545.127,Z 62.08,A -85,B 0,C 180,E1 -3501.847,E2 -3501.847} C_VEL
LIN {X 0,Y 545.205,Z 62.073,A -85,B 0,C 180,E1 -3504.823,E2 -3504.823} C_VEL
LIN {X 0,Y 545.196,Z 62.071,A -85,B 0,C 180,E1 -3507.784,E2 -3507.784} C_VEL
LIN {X 0,Y 545.21,Z 62.074,A -85,B 0,C 180,E1 -3510.739,E2 -3510.739} C_VEL
LIN {X 0,Y 545.169,Z 62.081,A -85,B 0,C 180,E1 -3512.956,E2 -3512.956} C_VEL
LIN {X 0,Y 545.177,Z 62.072,A -85,B 0,C 180,E1 -3515.919,E2 -3515.919} C_VEL
LIN {X 0,Y 545.118,Z 62.086,A -85,B 0,C 180,E1 -3518.9,E2 -3518.9} C_VEL
LIN {X 0,Y 545.132,Z 62.078,A -85,B 0,C 180,E1 -3521.904,E2 -3521.904} C_VEL
LIN {X 0,Y 545.083,Z 62.087,A -85,B 0,C 180,E1 -3524.944,E2 -3524.944} C_VEL
LIN {X 0,Y 545.077,Z 62.088,A -85,B 0,C 180,E1 -3528.026,E2 -3528.026} C_VEL
LIN {X 0,Y 545.092,Z 62.09,A -85,B 0,C 180,E1 -3530.372,E2 -3530.372} C_VEL
LIN {X 0,Y 545.088,Z 62.084,A -85,B 0,C 180,E1 -3533.559,E2 -3533.559} C_VEL
LIN {X 0,Y 545.077,Z 62.091,A -85,B 0,C 180,E1 -3536.001,E2 -3536.001} C_VEL
LIN {X 0,Y 545.087,Z 62.079,A -85,B 0,C 180,E1 -3538.749,E2 -3538.749} C_VEL
LIN {X 0,Y 545.075,Z 62.088,A -85,B 0,C 180,E1 -3541.683,E2 -3541.683} C_VEL
LIN {X 0,Y 545.079,Z 62.075,A -85,B 0,C 180,E1 -3544.563,E2 -3544.563} C_VEL
LIN {X 0,Y 545.037,Z 62.09,A -85,B 0,C 180,E1 -3547.304,E2 -3547.304} C_VEL
LIN {X 0,Y 545.071,Z 62.082,A -85,B 0,C 180,E1 -3550.142,E2 -3550.142} C_VEL
LIN {X 0,Y 545.058,Z 62.076,A -85,B 0,C 180,E1 -3552.697,E2 -3552.697} C_VEL
LIN {X 0,Y 545.059,Z 62.087,A -85,B 0,C 180,E1 -3555.167,E2 -3555.167} C_VEL
LIN {X 0,Y 545.079,Z 62.084,A -85,B 0,C 180,E1 -3557.898,E2 -3557.898} C_VEL
LIN {X 0,Y 545.081,Z 62.083,A -85,B 0,C 180,E1 -3560.819,E2 -3560.819} C_VEL
LIN {X 0,Y 545.054,Z 62.088,A -85,B 0,C 180,E1 -3563.621,E2 -3563.621} C_VEL
LIN {X 0,Y 545.069,Z 62.081,A -85,B 0,C 180,E1 -3566.329,E2 -3566.329} C_VEL
LIN {X 0,Y 545.065,Z 62.092,A -85,B 0,C 180,E1 -3568.953,E2 -3568.953} C_VEL
LIN {X 0,Y 545.101,Z 62.078,A -85,B 0,C 180,E1 -3571.508,E2 -3571.508} C_VEL
LIN {X 0,Y 545.093,Z 62.081,A -85,B 0,C 180,E1 -3574.491,E2 -3574.491} C_VEL
LIN {X 0,Y 545.043,Z 62.09,A -85,B 0,C 180,E1 -3577.243,E2 -3577.243} C_VEL
LIN {X 0,Y 545.119,Z 62.079,A -85,B 0,C 180,E1 -3580.415,E2 -3580.415} C_VEL
LIN {X 0,Y 545.072,Z 62.082,A -85,B 0,C 180,E1 -3583.522,E2 -3583.522} C_VEL
LIN {X 0,Y 545.094,Z 62.082,A -85,B 0,C 180,E1 -3585.82,E2 -3585.82} C_VEL
LIN {X 0,Y 545.117,Z 62.075,A -85,B 0,C 180,E1 -3588.85,E2 -3588.85} C_VEL
LIN {X 0,Y 545.128,Z 62.074,A -85,B 0,C 180,E1 -3591.847,E2 -3591.847} C_VEL
LIN {X 0,Y 545.203,Z 62.069,A -85,B 0,C 180,E1 -3594.823,E2 -3594.823} C_VEL
LIN {X 0,Y 545.196,Z 62.071,A -85,B 0,C 180,E1 -3597.784,E2 -3597.784} C_VEL
LIN {X 0,Y 545.213,Z 62.061,A -85,B 0,C 180,E1 -3600.739,E2 -3600.739} C_VEL
LIN {X 0,Y 545.17,Z 62.07,A -85,B 0,C 180,E1 -3602.956,E2 -3602.956} C_VEL
LIN {X 0,Y 545.172,Z 62.078,A -85,B 0,C 180,E1 -3605.92,E2 -3605.92} C_VEL
LIN {X 0,Y 545.117,Z 62.072,A -85,B 0,C 180,E1 -3608.9,E2 -3608.9} C_VEL
LIN {X 0,Y 545.136,Z 62.079,A -85,B 0,C 180,E1 -3611.905,E2 -3611.905} C_VEL
LIN {X 0,Y 545.086,Z 62.083,A -85,B 0,C 180,E1 -3614.944,E2 -3614.944} C_VEL
LIN {X 0,Y 545.078,Z 62.078,A -85,B 0,C 180,E1 -3618.026,E2 -3618.026} C_VEL
LIN {X 0,Y 545.096,Z 62.077,A -85,B 0,C 180,E1 -3620.372,E2 -3620.372} C_VEL
LIN {X 0,Y 545.092,Z 62.085,A -85,B 0,C 180,E1 -3623.559,E2 -3623.559} C_VEL
LIN {X 0,Y 545.08,Z 62.079,A -85,B 0,C 180,E1 -3626.001,E2 -3626.001} C_VEL
LIN {X 0,Y 545.09,Z 62.082,A -85,B 0,C 180,E1 -3628.748,E2 -3628.748} C_VEL
LIN {X 0,Y 545.059,Z 62.086,A -85,B 0,C 180,E1 -3631.679,E2 -3631.679} C_VEL
LIN {X 0,Y 545.077,Z 62.083,A -85,B 0,C 180,E1 -3634.564,E2 -3634.564} C_VEL
LIN {X 0,Y 545.038,Z 62.09,A -85,B 0,C 180,E1 -3637.304,E2 -3637.304} C_VEL
LIN {X 0,Y 545.07,Z 62.083,A -85,B 0,C 180,E1 -3640.143,E2 -3640.143} C_VEL
LIN {X 0,Y 545.08,Z 62.085,A -85,B 0,C 180,E1 -3643.107,E2 -3643.107} C_VEL
LIN {X 0,Y 545.05,Z 62.09,A -85,B 0,C 180,E1 -3646.227,E2 -3646.227} C_VEL
LIN {X 0,Y 545.083,Z 62.08,A -85,B 0,C 180,E1 -3648.886,E2 -3648.886} C_VEL
LIN {X 0,Y 545.081,Z 62.085,A -85,B 0,C 180,E1 -3650.818,E2 -3650.818} C_VEL
LIN {X 0,Y 545.051,Z 62.087,A -85,B 0,C 180,E1 -3653.62,E2 -3653.62} C_VEL
LIN {X 0,Y 545.07,Z 62.091,A -85,B 0,C 180,E1 -3656.329,E2 -3656.329} C_VEL
LIN {X 0,Y 545.069,Z 62.086,A -85,B 0,C 180,E1 -3658.952,E2 -3658.952} C_VEL
LIN {X 0,Y 545.105,Z 62.084,A -85,B 0,C 180,E1 -3661.508,E2 -3661.508} C_VEL
LIN {X 0,Y 545.116,Z 62.131,A -85,B 0,C 180,E1 -3664.488,E2 -3664.488} C_VEL
LIN {X 0,Y 545.968,Z 67.758,A -85,B 0,C 180,E1 -3665.674,E2 -3665.674} C_VEL
LIN {X 0,Y 545.678,Z 82.227,A -85,B 0,C 180,E1 -3668.465,E2 -3668.465} C_VEL
LIN {X 0,Y 545.431,Z 96.818,A -85,B 0,C 180,E1 -3671.208,E2 -3671.208} C_VEL
LIN {X 0,Y 545.298,Z 111.427,A -85,B 0,C 180,E1 -3673.913,E2 -3673.913} C_VEL
LIN {X 0,Y 545.126,Z 119.761,A -85,B 0,C 180,E1 -3675.426,E2 -3675.426} C_VEL
LIN {X 0,Y 546.363,Z 127.123,A -85,B 0,C 180,E1 -3675.587,E2 -3675.587} C_VEL
LIN {X 0,Y 546.222,Z 224.618,A -85,B 0,C 180,E1 -3676.893,E2 -3676.893} C_VEL
LIN {X 0,Y 546.09,Z 234.516,A -85,B 0,C 180,E1 -3677.102,E2 -3677.102} C_VEL
LIN {X 0,Y 545.995,Z 244.496,A -85,B 0,C 180,E1 -3677.407,E2 -3677.407} C_VEL
LIN {X 0,Y 545.84,Z 253.855,A -85,B 0,C 180,E1 -3677.781,E2 -3677.781} C_VEL
LIN {X 0,Y 545.642,Z 264.277,A -85,B 0,C 180,E1 -3678.312,E2 -3678.312} C_VEL
LIN {X 0,Y 545.496,Z 273.001,A -85,B 0,C 180,E1 -3678.857,E2 -3678.857} C_VEL
LIN {X 0,Y 545.333,Z 281.733,A -85,B 0,C 180,E1 -3679.512,E2 -3679.512} C_VEL
LIN {X 0,Y 545.17,Z 289.13,A -85,B 0,C 180,E1 -3680.165,E2 -3680.165} C_VEL
LIN {X 0,Y 545.046,Z 296.351,A -85,B 0,C 180,E1 -3680.912,E2 -3680.912} C_VEL
LIN {X 0,Y 544.944,Z 302.554,A -85,B 0,C 180,E1 -3681.658,E2 -3681.658} C_VEL
LIN {X 0,Y 544.829,Z 309.09,A -85,B 0,C 180,E1 -3682.589,E2 -3682.589} C_VEL
LIN {X 0,Y 544.741,Z 314.069,A -85,B 0,C 180,E1 -3683.425,E2 -3683.425} C_VEL
LIN {X 0,Y 544.735,Z 319.078,A -85,B 0,C 180,E1 -3684.447,E2 -3684.447} C_VEL
LIN {X 0,Y 544.66,Z 323.396,A -85,B 0,C 180,E1 -3685.56,E2 -3685.56} C_VEL
LIN {X 0,Y 544.669,Z 325.759,A -85,B 0,C 180,E1 -3686.301,E2 -3686.301} C_VEL
LIN {X 0,Y 544.65,Z 327.554,A -85,B 0,C 180,E1 -3687.041,E2 -3687.041} C_VEL
LIN {X 0,Y 544.547,Z 329.99,A -85,B 0,C 180,E1 -3688.521,E2 -3688.521} C_VEL
LIN {X 0,Y 544.544,Z 330.576,A -85,B 0,C 180,E1 -3689.261,E2 -3689.261} C_VEL
LIN {X 0,Y 544.544,Z 330.576,A -85,B 0,C 180,E1 -3690.739,E2 -3690.739} C_VEL
LIN {X 0,Y 544.547,Z 329.99,A -85,B 0,C 180,E1 -3691.479,E2 -3691.479} C_VEL
LIN {X 0,Y 544.65,Z 327.554,A -85,B 0,C 180,E1 -3692.959,E2 -3692.959} C_VEL
LIN {X 0,Y 544.684,Z 324.612,A -85,B 0,C 180,E1 -3694.069,E2 -3694.069} C_VEL
LIN {X 0,Y 544.653,Z 320.628,A -85,B 0,C 180,E1 -3695.182,E2 -3695.182} C_VEL
LIN {X 0,Y 544.737,Z 316.373,A -85,B 0,C 180,E1 -3696.127,E2 -3696.127} C_VEL
LIN {X 0,Y 544.783,Z 311.4,A -85,B 0,C 180,E1 -3697.04,E2 -3697.04} C_VEL
LIN {X 0,Y 544.892,Z 305.305,A -85,B 0,C 180,E1 -3697.97,E2 -3697.97} C_VEL
LIN {X 0,Y 544.975,Z 299.605,A -85,B 0,C 180,E1 -3698.715,E2 -3698.715} C_VEL
LIN {X 0,Y 545.123,Z 291.049,A -85,B 0,C 180,E1 -3699.648,E2 -3699.648} C_VEL
LIN {X 0,Y 545.308,Z 282.868,A -85,B 0,C 180,E1 -3700.395,E2 -3700.395} C_VEL
LIN {X 0,Y 545.475,Z 274.353,A -85,B 0,C 180,E1 -3701.049,E2 -3701.049} C_VEL
LIN {X 0,Y 545.639,Z 265.388,A -85,B 0,C 180,E1 -3701.624,E2 -3701.624} C_VEL
LIN {X 0,Y 545.849,Z 255.871,A -85,B 0,C 180,E1 -3702.124,E2 -3702.124} C_VEL
LIN {X 0,Y 545.941,Z 247.072,A -85,B 0,C 180,E1 -3702.499,E2 -3702.499} C_VEL
LIN {X 0,Y 546.072,Z 237.14,A -85,B 0,C 180,E1 -3702.827,E2 -3702.827} C_VEL
LIN {X 0,Y 546.186,Z 227.281,A -85,B 0,C 180,E1 -3703.061,E2 -3703.061} C_VEL
LIN {X 0,Y 546.327,Z 202.67,A -85,B 0,C 180,E1 -3703.412,E2 -3703.412} C_VEL
LIN {X 0,Y 546.361,Z 127.177,A -85,B 0,C 180,E1 -3704.412,E2 -3704.412} C_VEL
LIN {X 0,Y 545.134,Z 119.939,A -85,B 0,C 180,E1 -3704.562,E2 -3704.562} C_VEL
LIN {X 0,Y 545.161,Z 117.633,A -85,B 0,C 180,E1 -3704.941,E2 -3704.941} C_VEL
LIN {X 0,Y 545.375,Z 103.665,A -85,B 0,C 180,E1 -3707.521,E2 -3707.521} C_VEL
LIN {X 0,Y 545.586,Z 88.454,A -85,B 0,C 180,E1 -3710.353,E2 -3710.353} C_VEL
LIN {X 0,Y 545.902,Z 72.929,A -85,B 0,C 180,E1 -3713.321,E2 -3713.321} C_VEL
LIN {X 0,Y 545.9,Z 66.722,A -85,B 0,C 180,E1 -3714.531,E2 -3714.531} C_VEL
LIN {X 0,Y 545.11,Z 62.114,A -85,B 0,C 180,E1 -3715.511,E2 -3715.511} C_VEL
LIN {X 0,Y 545.105,Z 62.084,A -85,B 0,C 180,E1 -3718.492,E2 -3718.492} C_VEL
LIN {X 0,Y 545.069,Z 62.086,A -85,B 0,C 180,E1 -3721.048,E2 -3721.048} C_VEL
LIN {X 0,Y 545.07,Z 62.092,A -85,B 0,C 180,E1 -3723.671,E2 -3723.671} C_VEL
LIN {X 0,Y 545.075,Z 62.084,A -85,B 0,C 180,E1 -3726.926,E2 -3726.926} C_VEL
LIN {X 0,Y 545.067,Z 62.081,A -85,B 0,C 180,E1 -3730.142,E2 -3730.142} C_VEL
LIN {X 0,Y 545.08,Z 62.086,A -85,B 0,C 180,E1 -3733.106,E2 -3733.106} C_VEL
LIN {X 0,Y 545.05,Z 62.087,A -85,B 0,C 180,E1 -3736.226,E2 -3736.226} C_VEL
LIN {X 0,Y 545.083,Z 62.085,A -85,B 0,C 180,E1 -3738.885,E2 -3738.885} C_VEL
LIN {X 0,Y 545.085,Z 62.083,A -85,B 0,C 180,E1 -3740.818,E2 -3740.818} C_VEL
LIN {X 0,Y 545.044,Z 62.089,A -85,B 0,C 180,E1 -3743.619,E2 -3743.619} C_VEL
LIN {X 0,Y 545.068,Z 62.08,A -85,B 0,C 180,E1 -3746.328,E2 -3746.328} C_VEL
LIN {X 0,Y 545.067,Z 62.093,A -85,B 0,C 180,E1 -3748.952,E2 -3748.952} C_VEL
LIN {X 0,Y 545.102,Z 62.078,A -85,B 0,C 180,E1 -3751.507,E2 -3751.507} C_VEL
LIN {X 0,Y 545.096,Z 62.081,A -85,B 0,C 180,E1 -3754.491,E2 -3754.491} C_VEL
LIN {X 0,Y 545.045,Z 62.088,A -85,B 0,C 180,E1 -3757.242,E2 -3757.242} C_VEL
LIN {X 0,Y 545.121,Z 62.08,A -85,B 0,C 180,E1 -3760.415,E2 -3760.415} C_VEL
LIN {X 0,Y 545.074,Z 62.081,A -85,B 0,C 180,E1 -3763.521,E2 -3763.521} C_VEL
LIN {X 0,Y 545.096,Z 62.082,A -85,B 0,C 180,E1 -3765.82,E2 -3765.82} C_VEL
LIN {X 0,Y 545.119,Z 62.074,A -85,B 0,C 180,E1 -3768.849,E2 -3768.849} C_VEL
LIN {X 0,Y 545.129,Z 62.075,A -85,B 0,C 180,E1 -3771.847,E2 -3771.847} C_VEL
LIN {X 0,Y 545.203,Z 62.068,A -85,B 0,C 180,E1 -3774.823,E2 -3774.823} C_VEL
LIN {X 0,Y 545.198,Z 62.072,A -85,B 0,C 180,E1 -3777.783,E2 -3777.783} C_VEL
LIN {X 0,Y 545.212,Z 62.06,A -85,B 0,C 180,E1 -3780.738,E2 -3780.738} C_VEL
LIN {X 0,Y 545.17,Z 62.07,A -85,B 0,C 180,E1 -3782.955,E2 -3782.955} C_VEL
LIN {X 0,Y 545.171,Z 62.077,A -85,B 0,C 180,E1 -3785.919,E2 -3785.919} C_VEL
LIN {X 0,Y 545.117,Z 62.074,A -85,B 0,C 180,E1 -3788.9,E2 -3788.9} C_VEL
LIN {X 0,Y 545.134,Z 62.079,A -85,B 0,C 180,E1 -3791.904,E2 -3791.904} C_VEL
LIN {X 0,Y 545.085,Z 62.084,A -85,B 0,C 180,E1 -3794.943,E2 -3794.943} C_VEL
LIN {X 0,Y 545.078,Z 62.078,A -85,B 0,C 180,E1 -3798.025,E2 -3798.025} C_VEL
LIN {X 0,Y 545.094,Z 62.077,A -85,B 0,C 180,E1 -3800.372,E2 -3800.372} C_VEL
LIN {X 0,Y 545.09,Z 62.085,A -85,B 0,C 180,E1 -3803.558,E2 -3803.558} C_VEL
LIN {X 0,Y 545.078,Z 62.08,A -85,B 0,C 180,E1 -3806,E2 -3806} C_VEL
LIN {X 0,Y 545.087,Z 62.083,A -85,B 0,C 180,E1 -3808.748,E2 -3808.748} C_VEL
LIN {X 0,Y 545.076,Z 62.084,A -85,B 0,C 180,E1 -3811.682,E2 -3811.682} C_VEL
LIN {X 0,Y 545.08,Z 62.085,A -85,B 0,C 180,E1 -3814.563,E2 -3814.563} C_VEL
LIN {X 0,Y 545.063,Z 62.09,A -85,B 0,C 180,E1 -3817.004,E2 -3817.004} C_VEL
LIN {X 0,Y 544.353,Z 62.176,A -85,B 0,C 180,E1 -3817.62,E2 -3817.62} C_VEL
LIN {X 0,Y 541.486,Z 62.539,A -85,B 0,C 180,E1 -3818.621,E2 -3818.621} C_VEL
LIN {X 0,Y 539.103,Z 62.83,A -85,B 0,C 180,E1 -3819.427,E2 -3819.427} C_VEL
LIN {X 0,Y 538.102,Z 62.952,A -85,B 0,C 180,E1 -3820.049,E2 -3820.049} C_VEL
LIN {X 0,Y 538.031,Z 62.96,A -85,B 0,C 180,E1 -3820.259,E2 -3820.259} C_VEL
LIN {X 0,Y 538.023,Z 62.965,A -85,B 0,C 180,E1 -3822.987,E2 -3822.987} C_VEL
LIN {X 0,Y 538.021,Z 62.962,A -85,B 0,C 180,E1 -3825.926,E2 -3825.926} C_VEL
LIN {X 0,Y 538.049,Z 62.953,A -85,B 0,C 180,E1 -3829.252,E2 -3829.252} C_VEL
LIN {X 0,Y 537.991,Z 62.973,A -85,B 0,C 180,E1 -3832.122,E2 -3832.122} C_VEL
LIN {X 0,Y 538.017,Z 62.956,A -85,B 0,C 180,E1 -3834.917,E2 -3834.917} C_VEL
LIN {X 0,Y 538.024,Z 62.964,A -85,B 0,C 180,E1 -3837.618,E2 -3837.618} C_VEL
LIN {X 0,Y 538.015,Z 62.963,A -85,B 0,C 180,E1 -3840.239,E2 -3840.239} C_VEL
LIN {X 0,Y 538.063,Z 62.958,A -85,B 0,C 180,E1 -3842.796,E2 -3842.796} C_VEL
LIN {X 0,Y 538.046,Z 62.962,A -85,B 0,C 180,E1 -3845.293,E2 -3845.293} C_VEL
LIN {X 0,Y 538.012,Z 62.969,A -85,B 0,C 180,E1 -3848.042,E2 -3848.042} C_VEL
LIN {X 0,Y 538.035,Z 62.963,A -85,B 0,C 180,E1 -3850.94,E2 -3850.94} C_VEL
LIN {X 0,Y 538.023,Z 62.969,A -85,B 0,C 180,E1 -3853.299,E2 -3853.299} C_VEL
LIN {X 0,Y 538.061,Z 62.965,A -85,B 0,C 180,E1 -3855.631,E2 -3855.631} C_VEL
LIN {X 0,Y 538.075,Z 62.958,A -85,B 0,C 180,E1 -3858.702,E2 -3858.702} C_VEL
LIN {X 0,Y 538.084,Z 62.959,A -85,B 0,C 180,E1 -3861.74,E2 -3861.74} C_VEL
LIN {X 0,Y 538.163,Z 62.949,A -85,B 0,C 180,E1 -3864.755,E2 -3864.755} C_VEL
LIN {X 0,Y 538.167,Z 62.946,A -85,B 0,C 180,E1 -3867.755,E2 -3867.755} C_VEL
LIN {X 0,Y 538.18,Z 62.95,A -85,B 0,C 180,E1 -3870.748,E2 -3870.748} C_VEL
LIN {X 0,Y 538.135,Z 62.956,A -85,B 0,C 180,E1 -3872.994,E2 -3872.994} C_VEL
LIN {X 0,Y 538.131,Z 62.951,A -85,B 0,C 180,E1 -3875.997,E2 -3875.997} C_VEL
LIN {X 0,Y 538.069,Z 62.962,A -85,B 0,C 180,E1 -3879.018,E2 -3879.018} C_VEL
LIN {X 0,Y 538.081,Z 62.958,A -85,B 0,C 180,E1 -3882.063,E2 -3882.063} C_VEL
LIN {X 0,Y 538.043,Z 62.962,A -85,B 0,C 180,E1 -3885.144,E2 -3885.144} C_VEL
LIN {X 0,Y 538.029,Z 62.969,A -85,B 0,C 180,E1 -3888.27,E2 -3888.27} C_VEL
LIN {X 0,Y 538.036,Z 62.966,A -85,B 0,C 180,E1 -3890.651,E2 -3890.651} C_VEL
LIN {X 0,Y 538.021,Z 62.968,A -85,B 0,C 180,E1 -3893.887,E2 -3893.887} C_VEL
LIN {X 0,Y 538.039,Z 62.966,A -85,B 0,C 180,E1 -3896.367,E2 -3896.367} C_VEL
LIN {X 0,Y 538.028,Z 62.957,A -85,B 0,C 180,E1 -3898.934,E2 -3898.934} C_VEL
LIN {X 0,Y 538.025,Z 62.97,A -85,B 0,C 180,E1 -3901.891,E2 -3901.891} C_VEL
LIN {X 0,Y 538.029,Z 62.952,A -85,B 0,C 180,E1 -3904.621,E2 -3904.621} C_VEL
LIN {X 0,Y 538.005,Z 62.965,A -85,B 0,C 180,E1 -3907.171,E2 -3907.171} C_VEL
LIN {X 0,Y 538.027,Z 62.964,A -85,B 0,C 180,E1 -3909.796,E2 -3909.796} C_VEL
LIN {X 0,Y 538.009,Z 62.954,A -85,B 0,C 180,E1 -3912.787,E2 -3912.787} C_VEL
LIN {X 0,Y 538.028,Z 62.962,A -85,B 0,C 180,E1 -3915.141,E2 -3915.141} C_VEL
LIN {X 0,Y 538.037,Z 62.959,A -85,B 0,C 180,E1 -3918.228,E2 -3918.228} C_VEL
LIN {X 0,Y 538.036,Z 62.959,A -85,B 0,C 180,E1 -3920.414,E2 -3920.414} C_VEL
LIN {X 0,Y 538.027,Z 62.968,A -85,B 0,C 180,E1 -3923.068,E2 -3923.068} C_VEL
LIN {X 0,Y 538.025,Z 62.959,A -85,B 0,C 180,E1 -3925.828,E2 -3925.828} C_VEL
LIN {X 0,Y 538.008,Z 62.965,A -85,B 0,C 180,E1 -3928.499,E2 -3928.499} C_VEL
LIN {X 0,Y 538.058,Z 62.961,A -85,B 0,C 180,E1 -3931.1,E2 -3931.1} C_VEL
LIN {X 0,Y 538.04,Z 62.957,A -85,B 0,C 180,E1 -3933.634,E2 -3933.634} C_VEL
LIN {X 0,Y 538.021,Z 62.963,A -85,B 0,C 180,E1 -3936.118,E2 -3936.118} C_VEL
LIN {X 0,Y 538.038,Z 62.957,A -85,B 0,C 180,E1 -3939.349,E2 -3939.349} C_VEL
LIN {X 0,Y 538.053,Z 62.96,A -85,B 0,C 180,E1 -3942.517,E2 -3942.517} C_VEL
LIN {X 0,Y 538.063,Z 62.957,A -85,B 0,C 180,E1 -3945.631,E2 -3945.631} C_VEL
LIN {X 0,Y 538.076,Z 62.953,A -85,B 0,C 180,E1 -3948.702,E2 -3948.702} C_VEL
LIN {X 0,Y 538.085,Z 62.95,A -85,B 0,C 180,E1 -3951.74,E2 -3951.74} C_VEL
LIN {X 0,Y 538.161,Z 62.947,A -85,B 0,C 180,E1 -3954.755,E2 -3954.755} C_VEL
LIN {X 0,Y 538.168,Z 62.946,A -85,B 0,C 180,E1 -3957.755,E2 -3957.755} C_VEL
LIN {X 0,Y 538.183,Z 62.937,A -85,B 0,C 180,E1 -3960.749,E2 -3960.749} C_VEL
LIN {X 0,Y 538.136,Z 62.946,A -85,B 0,C 180,E1 -3962.995,E2 -3962.995} C_VEL
LIN {X 0,Y 538.125,Z 62.954,A -85,B 0,C 180,E1 -3965.998,E2 -3965.998} C_VEL
LIN {X 0,Y 538.068,Z 62.951,A -85,B 0,C 180,E1 -3969.018,E2 -3969.018} C_VEL
LIN {X 0,Y 538.084,Z 62.955,A -85,B 0,C 180,E1 -3972.063,E2 -3972.063} C_VEL
LIN {X 0,Y 538.046,Z 62.962,A -85,B 0,C 180,E1 -3975.144,E2 -3975.144} C_VEL
LIN {X 0,Y 538.031,Z 62.953,A -85,B 0,C 180,E1 -3978.271,E2 -3978.271} C_VEL
LIN {X 0,Y 538.04,Z 62.957,A -85,B 0,C 180,E1 -3980.652,E2 -3980.652} C_VEL
LIN {X 0,Y 538.026,Z 62.962,A -85,B 0,C 180,E1 -3983.888,E2 -3983.888} C_VEL
LIN {X 0,Y 538.043,Z 62.955,A -85,B 0,C 180,E1 -3986.367,E2 -3986.367} C_VEL
LIN {X 0,Y 538.032,Z 62.964,A -85,B 0,C 180,E1 -3988.934,E2 -3988.934} C_VEL
LIN {X 0,Y 538.011,Z 62.963,A -85,B 0,C 180,E1 -3991.887,E2 -3991.887} C_VEL
LIN {X 0,Y 538.026,Z 62.962,A -85,B 0,C 180,E1 -3994.62,E2 -3994.62} C_VEL
LIN {X 0,Y 538.006,Z 62.968,A -85,B 0,C 180,E1 -3997.17,E2 -3997.17} C_VEL
LIN {X 0,Y 538.027,Z 62.959,A -85,B 0,C 180,E1 -3999.797,E2 -3999.797} C_VEL
LIN {X 0,Y 538.02,Z 62.969,A -85,B 0,C 180,E1 -4002.786,E2 -4002.786} C_VEL
LIN {X 0,Y 538.02,Z 62.963,A -85,B 0,C 180,E1 -4005.927,E2 -4005.927} C_VEL
LIN {X 0,Y 538.032,Z 62.966,A -85,B 0,C 180,E1 -4008.227,E2 -4008.227} C_VEL
LIN {X 0,Y 538.013,Z 62.962,A -85,B 0,C 180,E1 -4011.17,E2 -4011.17} C_VEL
LIN {X 0,Y 538.026,Z 62.967,A -85,B 0,C 180,E1 -4014.085,E2 -4014.085} C_VEL
LIN {X 0,Y 538.033,Z 62.963,A -85,B 0,C 180,E1 -4016.728,E2 -4016.728} C_VEL
LIN {X 0,Y 538.029,Z 62.965,A -85,B 0,C 180,E1 -4019.556,E2 -4019.556} C_VEL
LIN {X 0,Y 538.047,Z 62.966,A -85,B 0,C 180,E1 -4021.951,E2 -4021.951} C_VEL
LIN {X 0,Y 538.064,Z 63.007,A -85,B 0,C 180,E1 -4024.324,E2 -4024.324} C_VEL
LIN {X 0,Y 539.022,Z 69.27,A -85,B 0,C 180,E1 -4025.667,E2 -4025.667} C_VEL
LIN {X 0,Y 538.679,Z 84.161,A -85,B 0,C 180,E1 -4028.574,E2 -4028.574} C_VEL
LIN {X 0,Y 538.437,Z 97.733,A -85,B 0,C 180,E1 -4031.153,E2 -4031.153} C_VEL
LIN {X 0,Y 538.251,Z 112.298,A -85,B 0,C 180,E1 -4033.891,E2 -4033.891} C_VEL
LIN {X 0,Y 538.078,Z 119.413,A -85,B 0,C 180,E1 -4035.217,E2 -4035.217} C_VEL
LIN {X 0,Y 538.539,Z 122.69,A -85,B 0,C 180,E1 -4035.316,E2 -4035.316} C_VEL
LIN {X 0,Y 539.617,Z 130.426,A -85,B 0,C 180,E1 -4035.45,E2 -4035.45} C_VEL
LIN {X 0,Y 539.306,Z 224.427,A -85,B 0,C 180,E1 -4036.722,E2 -4036.722} C_VEL
LIN {X 0,Y 539.159,Z 234.325,A -85,B 0,C 180,E1 -4036.934,E2 -4036.934} C_VEL
LIN {X 0,Y 539.053,Z 244.305,A -85,B 0,C 180,E1 -4037.243,E2 -4037.243} C_VEL
LIN {X 0,Y 538.909,Z 253.665,A -85,B 0,C 180,E1 -4037.622,E2 -4037.622} C_VEL
LIN {X 0,Y 538.684,Z 263.434,A -85,B 0,C 180,E1 -4038.12,E2 -4038.12} C_VEL
LIN {X 0,Y 538.496,Z 272.809,A -85,B 0,C 180,E1 -4038.71,E2 -4038.71} C_VEL
LIN {X 0,Y 538.328,Z 281.541,A -85,B 0,C 180,E1 -4039.374,E2 -4039.374} C_VEL
LIN {X 0,Y 538.149,Z 288.938,A -85,B 0,C 180,E1 -4040.035,E2 -4040.035} C_VEL
LIN {X 0,Y 538.001,Z 296.159,A -85,B 0,C 180,E1 -4040.792,E2 -4040.792} C_VEL
LIN {X 0,Y 537.898,Z 302.362,A -85,B 0,C 180,E1 -4041.548,E2 -4041.548} C_VEL
LIN {X 0,Y 537.744,Z 308.898,A -85,B 0,C 180,E1 -4042.49,E2 -4042.49} C_VEL
LIN {X 0,Y 537.64,Z 314.446,A -85,B 0,C 180,E1 -4043.45,E2 -4043.45} C_VEL
LIN {X 0,Y 537.648,Z 318.887,A -85,B 0,C 180,E1 -4044.374,E2 -4044.374} C_VEL
LIN {X 0,Y 537.556,Z 323.205,A -85,B 0,C 180,E1 -4045.501,E2 -4045.501} C_VEL
LIN {X 0,Y 537.591,Z 325.569,A -85,B 0,C 180,E1 -4046.252,E2 -4046.252} C_VEL
LIN {X 0,Y 537.551,Z 327.363,A -85,B 0,C 180,E1 -4047.002,E2 -4047.002} C_VEL
LIN {X 0,Y 537.452,Z 329.799,A -85,B 0,C 180,E1 -4048.501,E2 -4048.501} C_VEL
LIN {X 0,Y 537.446,Z 330.386,A -85,B 0,C 180,E1 -4049.251,E2 -4049.251} C_VEL
LIN {X 0,Y 537.446,Z 330.386,A -85,B 0,C 180,E1 -4050.749,E2 -4050.749} C_VEL
LIN {X 0,Y 537.452,Z 329.799,A -85,B 0,C 180,E1 -4051.499,E2 -4051.499} C_VEL
LIN {X 0,Y 537.551,Z 327.363,A -85,B 0,C 180,E1 -4052.998,E2 -4052.998} C_VEL
LIN {X 0,Y 537.604,Z 324.421,A -85,B 0,C 180,E1 -4054.123,E2 -4054.123} C_VEL
LIN {X 0,Y 537.586,Z 320.438,A -85,B 0,C 180,E1 -4055.251,E2 -4055.251} C_VEL
LIN {X 0,Y 537.619,Z 315.669,A -85,B 0,C 180,E1 -4056.309,E2 -4056.309} C_VEL
LIN {X 0,Y 537.752,Z 310.054,A -85,B 0,C 180,E1 -4057.321,E2 -4057.321} C_VEL
LIN {X 0,Y 537.869,Z 303.738,A -85,B 0,C 180,E1 -4058.264,E2 -4058.264} C_VEL
LIN {X 0,Y 537.948,Z 297.786,A -85,B 0,C 180,E1 -4059.02,E2 -4059.02} C_VEL
LIN {X 0,Y 538.08,Z 290.857,A -85,B 0,C 180,E1 -4059.776,E2 -4059.776} C_VEL
LIN {X 0,Y 538.304,Z 282.677,A -85,B 0,C 180,E1 -4060.532,E2 -4060.532} C_VEL
LIN {X 0,Y 538.492,Z 274.162,A -85,B 0,C 180,E1 -4061.194,E2 -4061.194} C_VEL
LIN {X 0,Y 538.639,Z 265.196,A -85,B 0,C 180,E1 -4061.778,E2 -4061.778} C_VEL
LIN {X 0,Y 538.883,Z 255.68,A -85,B 0,C 180,E1 -4062.283,E2 -4062.283} C_VEL
LIN {X 0,Y 539.004,Z 246.881,A -85,B 0,C 180,E1 -4062.663,E2 -4062.663} C_VEL
LIN {X 0,Y 539.169,Z 236.95,A -85,B 0,C 180,E1 -4062.994,E2 -4062.994} C_VEL
LIN {X 0,Y 539.277,Z 227.091,A -85,B 0,C 180,E1 -4063.231,E2 -4063.231} C_VEL
LIN {X 0,Y 539.439,Z 202.48,A -85,B 0,C 180,E1 -4063.587,E2 -4063.587} C_VEL
LIN {X 0,Y 539.454,Z 127.955,A -85,B 0,C 180,E1 -4064.588,E2 -4064.588} C_VEL
LIN {X 0,Y 538.124,Z 119.845,A -85,B 0,C 180,E1 -4064.75,E2 -4064.75} C_VEL
LIN {X 0,Y 538.101,Z 118.819,A -85,B 0,C 180,E1 -4064.873,E2 -4064.873} C_VEL
LIN {X 0,Y 538.373,Z 104.131,A -85,B 0,C 180,E1 -4067.644,E2 -4067.644} C_VEL
LIN {X 0,Y 538.591,Z 90.21,A -85,B 0,C 180,E1 -4070.269,E2 -4070.269} C_VEL
LIN {X 0,Y 538.955,Z 73.831,A -85,B 0,C 180,E1 -4073.436,E2 -4073.436} C_VEL
LIN {X 0,Y 538.9,Z 67.634,A -85,B 0,C 180,E1 -4074.666,E2 -4074.666} C_VEL
LIN {X 0,Y 538.071,Z 62.991,A -85,B 0,C 180,E1 -4075.683,E2 -4075.683} C_VEL
LIN {X 0,Y 538.047,Z 62.966,A -85,B 0,C 180,E1 -4078.049,E2 -4078.049} C_VEL
LIN {X 0,Y 538.023,Z 62.965,A -85,B 0,C 180,E1 -4080.627,E2 -4080.627} C_VEL
LIN {X 0,Y 538.048,Z 62.961,A -85,B 0,C 180,E1 -4083.283,E2 -4083.283} C_VEL
LIN {X 0,Y 538.025,Z 62.967,A -85,B 0,C 180,E1 -4086.002,E2 -4086.002} C_VEL
LIN {X 0,Y 538.014,Z 62.963,A -85,B 0,C 180,E1 -4088.83,E2 -4088.83} C_VEL
LIN {X 0,Y 538.032,Z 62.966,A -85,B 0,C 180,E1 -4091.773,E2 -4091.773} C_VEL
LIN {X 0,Y 538.006,Z 62.965,A -85,B 0,C 180,E1 -4094.862,E2 -4094.862} C_VEL
LIN {X 0,Y 538.021,Z 62.969,A -85,B 0,C 180,E1 -4097.214,E2 -4097.214} C_VEL
LIN {X 0,Y 538.027,Z 62.959,A -85,B 0,C 180,E1 -4100.203,E2 -4100.203} C_VEL
LIN {X 0,Y 538.026,Z 62.969,A -85,B 0,C 180,E1 -4103.067,E2 -4103.067} C_VEL
LIN {X 0,Y 538.025,Z 62.957,A -85,B 0,C 180,E1 -4105.827,E2 -4105.827} C_VEL
LIN {X 0,Y 538.01,Z 62.965,A -85,B 0,C 180,E1 -4108.498,E2 -4108.498} C_VEL
LIN {X 0,Y 538.061,Z 62.96,A -85,B 0,C 180,E1 -4111.1,E2 -4111.1} C_VEL
LIN {X 0,Y 538.043,Z 62.955,A -85,B 0,C 180,E1 -4113.633,E2 -4113.633} C_VEL
LIN {X 0,Y 538.024,Z 62.962,A -85,B 0,C 180,E1 -4116.118,E2 -4116.118} C_VEL
LIN {X 0,Y 538.04,Z 62.957,A -85,B 0,C 180,E1 -4119.348,E2 -4119.348} C_VEL
LIN {X 0,Y 538.055,Z 62.959,A -85,B 0,C 180,E1 -4122.517,E2 -4122.517} C_VEL
LIN {X 0,Y 538.065,Z 62.956,A -85,B 0,C 180,E1 -4125.63,E2 -4125.63} C_VEL
LIN {X 0,Y 538.078,Z 62.952,A -85,B 0,C 180,E1 -4128.701,E2 -4128.701} C_VEL
LIN {X 0,Y 538.086,Z 62.95,A -85,B 0,C 180,E1 -4131.739,E2 -4131.739} C_VEL
LIN {X 0,Y 538.161,Z 62.946,A -85,B 0,C 180,E1 -4134.755,E2 -4134.755} C_VEL
LIN {X 0,Y 538.169,Z 62.947,A -85,B 0,C 180,E1 -4137.754,E2 -4137.754} C_VEL
LIN {X 0,Y 538.182,Z 62.935,A -85,B 0,C 180,E1 -4140.748,E2 -4140.748} C_VEL
LIN {X 0,Y 538.137,Z 62.946,A -85,B 0,C 180,E1 -4142.994,E2 -4142.994} C_VEL
LIN {X 0,Y 538.124,Z 62.953,A -85,B 0,C 180,E1 -4145.997,E2 -4145.997} C_VEL
LIN {X 0,Y 538.068,Z 62.952,A -85,B 0,C 180,E1 -4149.017,E2 -4149.017} C_VEL
LIN {X 0,Y 538.083,Z 62.955,A -85,B 0,C 180,E1 -4152.062,E2 -4152.062} C_VEL
LIN {X 0,Y 538.044,Z 62.964,A -85,B 0,C 180,E1 -4155.143,E2 -4155.143} C_VEL
LIN {X 0,Y 538.03,Z 62.955,A -85,B 0,C 180,E1 -4158.27,E2 -4158.27} C_VEL
LIN {X 0,Y 538.038,Z 62.957,A -85,B 0,C 180,E1 -4160.651,E2 -4160.651} C_VEL
LIN {X 0,Y 538.023,Z 62.962,A -85,B 0,C 180,E1 -4163.887,E2 -4163.887} C_VEL
LIN {X 0,Y 538.04,Z 62.957,A -85,B 0,C 180,E1 -4166.366,E2 -4166.366} C_VEL
LIN {X 0,Y 538.029,Z 62.965,A -85,B 0,C 180,E1 -4168.933,E2 -4168.933} C_VEL
LIN {X 0,Y 538.025,Z 62.961,A -85,B 0,C 180,E1 -4171.89,E2 -4171.89} C_VEL
LIN {X 0,Y 538.03,Z 62.964,A -85,B 0,C 180,E1 -4174.621,E2 -4174.621} C_VEL
LIN {X 0,Y 538.005,Z 62.967,A -85,B 0,C 180,E1 -4177.17,E2 -4177.17} C_VEL
LIN {X 0,Y 538.031,Z 62.96,A -85,B 0,C 180,E1 -4180.259,E2 -4180.259} C_VEL
LIN {X 0,Y 537.391,Z 63.044,A -85,B 0,C 180,E1 -4180.885,E2 -4180.885} C_VEL
LIN {X 0,Y 534.536,Z 63.399,A -85,B 0,C 180,E1 -4181.899,E2 -4181.899} C_VEL
LIN {X 0,Y 532.101,Z 63.706,A -85,B 0,C 180,E1 -4182.716,E2 -4182.716} C_VEL
LIN {X 0,Y 531.048,Z 63.832,A -85,B 0,C 180,E1 -4183.347,E2 -4183.347} C_VEL
LIN {X 0,Y 530.959,Z 63.842,A -85,B 0,C 180,E1 -4183.561,E2 -4183.561} C_VEL
LIN {X 0,Y 530.956,Z 63.839,A -85,B 0,C 180,E1 -4186.505,E2 -4186.505} C_VEL
LIN {X 0,Y 530.986,Z 63.834,A -85,B 0,C 180,E1 -4188.975,E2 -4188.975} C_VEL
LIN {X 0,Y 530.956,Z 63.843,A -85,B 0,C 180,E1 -4191.529,E2 -4191.529} C_VEL
LIN {X 0,Y 530.979,Z 63.837,A -85,B 0,C 180,E1 -4194.382,E2 -4194.382} C_VEL
LIN {X 0,Y 530.968,Z 63.84,A -85,B 0,C 180,E1 -4197.134,E2 -4197.134} C_VEL
LIN {X 0,Y 530.967,Z 63.846,A -85,B 0,C 180,E1 -4199.803,E2 -4199.803} C_VEL
LIN {X 0,Y 531.013,Z 63.838,A -85,B 0,C 180,E1 -4202.467,E2 -4202.467} C_VEL
LIN {X 0,Y 531.003,Z 63.837,A -85,B 0,C 180,E1 -4204.942,E2 -4204.942} C_VEL
LIN {X 0,Y 530.968,Z 63.844,A -85,B 0,C 180,E1 -4208.247,E2 -4208.247} C_VEL
LIN {X 0,Y 530.992,Z 63.839,A -85,B 0,C 180,E1 -4210.677,E2 -4210.677} C_VEL
LIN {X 0,Y 530.983,Z 63.843,A -85,B 0,C 180,E1 -4213.071,E2 -4213.071} C_VEL
LIN {X 0,Y 531.038,Z 63.841,A -85,B 0,C 180,E1 -4215.436,E2 -4215.436} C_VEL
LIN {X 0,Y 531.034,Z 63.835,A -85,B 0,C 180,E1 -4218.55,E2 -4218.55} C_VEL
LIN {X 0,Y 531.054,Z 63.836,A -85,B 0,C 180,E1 -4221.629,E2 -4221.629} C_VEL
LIN {X 0,Y 531.122,Z 63.826,A -85,B 0,C 180,E1 -4224.685,E2 -4224.685} C_VEL
LIN {X 0,Y 531.139,Z 63.822,A -85,B 0,C 180,E1 -4227.725,E2 -4227.725} C_VEL
LIN {X 0,Y 531.151,Z 63.825,A -85,B 0,C 180,E1 -4230.758,E2 -4230.758} C_VEL
LIN {X 0,Y 531.102,Z 63.832,A -85,B 0,C 180,E1 -4233.034,E2 -4233.034} C_VEL
LIN {X 0,Y 531.089,Z 63.828,A -85,B 0,C 180,E1 -4236.077,E2 -4236.077} C_VEL
LIN {X 0,Y 531.029,Z 63.838,A -85,B 0,C 180,E1 -4239.138,E2 -4239.138} C_VEL
LIN {X 0,Y 531.038,Z 63.838,A -85,B 0,C 180,E1 -4242.225,E2 -4242.225} C_VEL
LIN {X 0,Y 530.993,Z 63.84,A -85,B 0,C 180,E1 -4245.35,E2 -4245.35} C_VEL
LIN {X 0,Y 530.988,Z 63.846,A -85,B 0,C 180,E1 -4248.521,E2 -4248.521} C_VEL
LIN {X 0,Y 530.997,Z 63.84,A -85,B 0,C 180,E1 -4250.938,E2 -4250.938} C_VEL
LIN {X 0,Y 530.977,Z 63.848,A -85,B 0,C 180,E1 -4254.225,E2 -4254.225} C_VEL
LIN {X 0,Y 531.003,Z 63.839,A -85,B 0,C 180,E1 -4256.744,E2 -4256.744} C_VEL
LIN {X 0,Y 530.979,Z 63.836,A -85,B 0,C 180,E1 -4259.323,E2 -4259.323} C_VEL
LIN {X 0,Y 530.977,Z 63.845,A -85,B 0,C 180,E1 -4262.103,E2 -4262.103} C_VEL
LIN {X 0,Y 530.986,Z 63.828,A -85,B 0,C 180,E1 -4264.854,E2 -4264.854} C_VEL
LIN {X 0,Y 530.964,Z 63.846,A -85,B 0,C 180,E1 -4267.508,E2 -4267.508} C_VEL
LIN {X 0,Y 530.981,Z 63.834,A -85,B 0,C 180,E1 -4270.433,E2 -4270.433} C_VEL
LIN {X 0,Y 530.947,Z 63.837,A -85,B 0,C 180,E1 -4273.28,E2 -4273.28} C_VEL
LIN {X 0,Y 530.985,Z 63.846,A -85,B 0,C 180,E1 -4275.621,E2 -4275.621} C_VEL
LIN {X 0,Y 531.004,Z 63.835,A -85,B 0,C 180,E1 -4278.566,E2 -4278.566} C_VEL
LIN {X 0,Y 530.957,Z 63.848,A -85,B 0,C 180,E1 -4281.53,E2 -4281.53} C_VEL
LIN {X 0,Y 530.98,Z 63.838,A -85,B 0,C 180,E1 -4284.383,E2 -4284.383} C_VEL
LIN {X 0,Y 530.968,Z 63.846,A -85,B 0,C 180,E1 -4287.134,E2 -4287.134} C_VEL
LIN {X 0,Y 530.967,Z 63.841,A -85,B 0,C 180,E1 -4289.803,E2 -4289.803} C_VEL
LIN {X 0,Y 531.014,Z 63.833,A -85,B 0,C 180,E1 -4292.467,E2 -4292.467} C_VEL
LIN {X 0,Y 531.004,Z 63.843,A -85,B 0,C 180,E1 -4294.943,E2 -4294.943} C_VEL
LIN {X 0,Y 530.97,Z 63.842,A -85,B 0,C 180,E1 -4298.247,E2 -4298.247} C_VEL
LIN {X 0,Y 530.994,Z 63.837,A -85,B 0,C 180,E1 -4300.678,E2 -4300.678} C_VEL
LIN {X 0,Y 530.985,Z 63.84,A -85,B 0,C 180,E1 -4303.071,E2 -4303.071} C_VEL
LIN {X 0,Y 531.018,Z 63.834,A -85,B 0,C 180,E1 -4305.436,E2 -4305.436} C_VEL
LIN {X 0,Y 531.048,Z 63.831,A -85,B 0,C 180,E1 -4308.55,E2 -4308.55} C_VEL
LIN {X 0,Y 531.055,Z 63.825,A -85,B 0,C 180,E1 -4311.63,E2 -4311.63} C_VEL
LIN {X 0,Y 531.12,Z 63.824,A -85,B 0,C 180,E1 -4314.686,E2 -4314.686} C_VEL
LIN {X 0,Y 531.14,Z 63.821,A -85,B 0,C 180,E1 -4317.725,E2 -4317.725} C_VEL
LIN {X 0,Y 531.153,Z 63.812,A -85,B 0,C 180,E1 -4320.759,E2 -4320.759} C_VEL
LIN {X 0,Y 531.103,Z 63.822,A -85,B 0,C 180,E1 -4323.035,E2 -4323.035} C_VEL
LIN {X 0,Y 531.085,Z 63.83,A -85,B 0,C 180,E1 -4326.077,E2 -4326.077} C_VEL
LIN {X 0,Y 531.029,Z 63.828,A -85,B 0,C 180,E1 -4329.139,E2 -4329.139} C_VEL
LIN {X 0,Y 531.041,Z 63.831,A -85,B 0,C 180,E1 -4332.225,E2 -4332.225} C_VEL
LIN {X 0,Y 530.996,Z 63.843,A -85,B 0,C 180,E1 -4335.35,E2 -4335.35} C_VEL
LIN {X 0,Y 530.99,Z 63.83,A -85,B 0,C 180,E1 -4338.522,E2 -4338.522} C_VEL
LIN {X 0,Y 531.001,Z 63.836,A -85,B 0,C 180,E1 -4340.938,E2 -4340.938} C_VEL
LIN {X 0,Y 530.981,Z 63.838,A -85,B 0,C 180,E1 -4344.225,E2 -4344.225} C_VEL
LIN {X 0,Y 531.002,Z 63.834,A -85,B 0,C 180,E1 -4346.744,E2 -4346.744} C_VEL
LIN {X 0,Y 530.983,Z 63.844,A -85,B 0,C 180,E1 -4349.323,E2 -4349.323} C_VEL
LIN {X 0,Y 530.966,Z 63.84,A -85,B 0,C 180,E1 -4352.101,E2 -4352.101} C_VEL
LIN {X 0,Y 530.981,Z 63.841,A -85,B 0,C 180,E1 -4354.853,E2 -4354.853} C_VEL
LIN {X 0,Y 530.967,Z 63.842,A -85,B 0,C 180,E1 -4357.508,E2 -4357.508} C_VEL
LIN {X 0,Y 530.983,Z 63.841,A -85,B 0,C 180,E1 -4360.433,E2 -4360.433} C_VEL
LIN {X 0,Y 530.962,Z 63.842,A -85,B 0,C 180,E1 -4363.281,E2 -4363.281} C_VEL
LIN {X 0,Y 530.977,Z 63.839,A -85,B 0,C 180,E1 -4365.623,E2 -4365.623} C_VEL
LIN {X 0,Y 530.995,Z 63.839,A -85,B 0,C 180,E1 -4368.565,E2 -4368.565} C_VEL
LIN {X 0,Y 530.957,Z 63.841,A -85,B 0,C 180,E1 -4371.529,E2 -4371.529} C_VEL
LIN {X 0,Y 530.978,Z 63.842,A -85,B 0,C 180,E1 -4374.382,E2 -4374.382} C_VEL
LIN {X 0,Y 530.969,Z 63.841,A -85,B 0,C 180,E1 -4377.134,E2 -4377.134} C_VEL
LIN {X 0,Y 530.973,Z 63.847,A -85,B 0,C 180,E1 -4379.803,E2 -4379.803} C_VEL
LIN {X 0,Y 531.018,Z 63.839,A -85,B 0,C 180,E1 -4382.467,E2 -4382.467} C_VEL
LIN {X 0,Y 531.024,Z 63.879,A -85,B 0,C 180,E1 -4384.154,E2 -4384.154} C_VEL
LIN {X 0,Y 532.008,Z 69.53,A -85,B 0,C 180,E1 -4385.402,E2 -4385.402} C_VEL
LIN {X 0,Y 531.787,Z 81.011,A -85,B 0,C 180,E1 -4387.685,E2 -4387.685} C_VEL
LIN {X 0,Y 531.477,Z 96.558,A -85,B 0,C 180,E1 -4390.696,E2 -4390.696} C_VEL
LIN {X 0,Y 531.231,Z 112.137,A -85,B 0,C 180,E1 -4393.672,E2 -4393.672} C_VEL
LIN {X 0,Y 531.053,Z 119.452,A -85,B 0,C 180,E1 -4395.037,E2 -4395.037} C_VEL
LIN {X 0,Y 532.748,Z 130.469,A -85,B 0,C 180,E1 -4395.262,E2 -4395.262} C_VEL
LIN {X 0,Y 532.416,Z 224.237,A -85,B 0,C 180,E1 -4396.547,E2 -4396.547} C_VEL
LIN {X 0,Y 532.24,Z 235.009,A -85,B 0,C 180,E1 -4396.785,E2 -4396.785} C_VEL
LIN {X 0,Y 532.122,Z 244.114,A -85,B 0,C 180,E1 -4397.073,E2 -4397.073} C_VEL
LIN {X 0,Y 531.949,Z 253.473,A -85,B 0,C 180,E1 -4397.457,E2 -4397.457} C_VEL
LIN {X 0,Y 531.707,Z 263.762,A -85,B 0,C 180,E1 -4397.993,E2 -4397.993} C_VEL
LIN {X 0,Y 531.502,Z 272.618,A -85,B 0,C 180,E1 -4398.56,E2 -4398.56} C_VEL
LIN {X 0,Y 531.33,Z 281.35,A -85,B 0,C 180,E1 -4399.232,E2 -4399.232} C_VEL
LIN {X 0,Y 531.139,Z 288.747,A -85,B 0,C 180,E1 -4399.903,E2 -4399.903} C_VEL
LIN {X 0,Y 530.968,Z 295.968,A -85,B 0,C 180,E1 -4400.669,E2 -4400.669} C_VEL
LIN {X 0,Y 530.851,Z 302.171,A -85,B 0,C 180,E1 -4401.435,E2 -4401.435} C_VEL
LIN {X 0,Y 530.675,Z 308.707,A -85,B 0,C 180,E1 -4402.39,E2 -4402.39} C_VEL
LIN {X 0,Y 530.578,Z 313.207,A -85,B 0,C 180,E1 -4403.153,E2 -4403.153} C_VEL
LIN {X 0,Y 530.564,Z 318.696,A -85,B 0,C 180,E1 -4404.298,E2 -4404.298} C_VEL
LIN {X 0,Y 530.454,Z 323.014,A -85,B 0,C 180,E1 -4405.441,E2 -4405.441} C_VEL
LIN {X 0,Y 530.516,Z 325.379,A -85,B 0,C 180,E1 -4406.202,E2 -4406.202} C_VEL
LIN {X 0,Y 530.457,Z 327.172,A -85,B 0,C 180,E1 -4406.962,E2 -4406.962} C_VEL
LIN {X 0,Y 530.362,Z 329.609,A -85,B 0,C 180,E1 -4408.481,E2 -4408.481} C_VEL
LIN {X 0,Y 530.349,Z 330.196,A -85,B 0,C 180,E1 -4409.241,E2 -4409.241} C_VEL
LIN {X 0,Y 530.349,Z 330.196,A -85,B 0,C 180,E1 -4410.759,E2 -4410.759} C_VEL
LIN {X 0,Y 530.362,Z 329.609,A -85,B 0,C 180,E1 -4411.519,E2 -4411.519} C_VEL
LIN {X 0,Y 530.457,Z 327.172,A -85,B 0,C 180,E1 -4413.038,E2 -4413.038} C_VEL
LIN {X 0,Y 530.522,Z 324.231,A -85,B 0,C 180,E1 -4414.178,E2 -4414.178} C_VEL
LIN {X 0,Y 530.519,Z 320.248,A -85,B 0,C 180,E1 -4415.321,E2 -4415.321} C_VEL
LIN {X 0,Y 530.526,Z 316.011,A -85,B 0,C 180,E1 -4416.288,E2 -4416.288} C_VEL
LIN {X 0,Y 530.665,Z 311.018,A -85,B 0,C 180,E1 -4417.228,E2 -4417.228} C_VEL
LIN {X 0,Y 530.775,Z 304.923,A -85,B 0,C 180,E1 -4418.183,E2 -4418.183} C_VEL
LIN {X 0,Y 530.874,Z 299.222,A -85,B 0,C 180,E1 -4418.949,E2 -4418.949} C_VEL
LIN {X 0,Y 531.045,Z 290.666,A -85,B 0,C 180,E1 -4419.907,E2 -4419.907} C_VEL
LIN {X 0,Y 531.307,Z 282.486,A -85,B 0,C 180,E1 -4420.672,E2 -4420.672} C_VEL
LIN {X 0,Y 531.504,Z 273.971,A -85,B 0,C 180,E1 -4421.343,E2 -4421.343} C_VEL
LIN {X 0,Y 531.663,Z 265.016,A -85,B 0,C 180,E1 -4421.934,E2 -4421.934} C_VEL
LIN {X 0,Y 531.928,Z 255.489,A -85,B 0,C 180,E1 -4422.446,E2 -4422.446} C_VEL
LIN {X 0,Y 532.083,Z 246.691,A -85,B 0,C 180,E1 -4422.83,E2 -4422.83} C_VEL
LIN {X 0,Y 532.257,Z 236.759,A -85,B 0,C 180,E1 -4423.166,E2 -4423.166} C_VEL
LIN {X 0,Y 532.363,Z 226.9,A -85,B 0,C 180,E1 -4423.406,E2 -4423.406} C_VEL
LIN {X 0,Y 532.562,Z 202.29,A -85,B 0,C 180,E1 -4423.766,E2 -4423.766} C_VEL
LIN {X 0,Y 532.699,Z 129.385,A -85,B 0,C 180,E1 -4424.755,E2 -4424.755} C_VEL
LIN {X 0,Y 531.101,Z 119.583,A -85,B 0,C 180,E1 -4424.953,E2 -4424.953} C_VEL
LIN {X 0,Y 531.06,Z 118.408,A -85,B 0,C 180,E1 -4425.121,E2 -4425.121} C_VEL
LIN {X 0,Y 531.366,Z 104.611,A -85,B 0,C 180,E1 -4427.769,E2 -4427.769} C_VEL
LIN {X 0,Y 531.617,Z 89.239,A -85,B 0,C 180,E1 -4430.71,E2 -4430.71} C_VEL
LIN {X 0,Y 531.984,Z 73.707,A -85,B 0,C 180,E1 -4433.762,E2 -4433.762} C_VEL
LIN {X 0,Y 531.879,Z 68.541,A -85,B 0,C 180,E1 -4434.809,E2 -4434.809} C_VEL
LIN {X 0,Y 531.033,Z 63.862,A -85,B 0,C 180,E1 -4435.859,E2 -4435.859} C_VEL
LIN {X 0,Y 531.002,Z 63.842,A -85,B 0,C 180,E1 -4438.455,E2 -4438.455} C_VEL
LIN {X 0,Y 530.96,Z 63.845,A -85,B 0,C 180,E1 -4441.079,E2 -4441.079} C_VEL
LIN {X 0,Y 530.992,Z 63.847,A -85,B 0,C 180,E1 -4443.772,E2 -4443.772} C_VEL
LIN {X 0,Y 530.967,Z 63.841,A -85,B 0,C 180,E1 -4446.557,E2 -4446.557} C_VEL
LIN {X 0,Y 530.979,Z 63.838,A -85,B 0,C 180,E1 -4449.853,E2 -4449.853} C_VEL
LIN {X 0,Y 530.979,Z 63.839,A -85,B 0,C 180,E1 -4452.456,E2 -4452.456} C_VEL
LIN {X 0,Y 530.977,Z 63.845,A -85,B 0,C 180,E1 -4455.622,E2 -4455.622} C_VEL
LIN {X 0,Y 530.995,Z 63.838,A -85,B 0,C 180,E1 -4458.564,E2 -4458.564} C_VEL
LIN {X 0,Y 530.961,Z 63.846,A -85,B 0,C 180,E1 -4461.529,E2 -4461.529} C_VEL
LIN {X 0,Y 530.959,Z 63.841,A -85,B 0,C 180,E1 -4464.38,E2 -4464.38} C_VEL
LIN {X 0,Y 530.968,Z 63.847,A -85,B 0,C 180,E1 -4467.133,E2 -4467.133} C_VEL
LIN {X 0,Y 530.97,Z 63.84,A -85,B 0,C 180,E1 -4469.803,E2 -4469.803} C_VEL
LIN {X 0,Y 531.014,Z 63.835,A -85,B 0,C 180,E1 -4472.467,E2 -4472.467} C_VEL
LIN {X 0,Y 531.007,Z 63.841,A -85,B 0,C 180,E1 -4474.942,E2 -4474.942} C_VEL
LIN {X 0,Y 530.973,Z 63.842,A -85,B 0,C 180,E1 -4478.246,E2 -4478.246} C_VEL
LIN {X 0,Y 530.995,Z 63.836,A -85,B 0,C 180,E1 -4480.677,E2 -4480.677} C_VEL
LIN {X 0,Y 530.986,Z 63.837,A -85,B 0,C 180,E1 -4483.071,E2 -4483.071} C_VEL
LIN {X 0,Y 531.02,Z 63.833,A -85,B 0,C 180,E1 -4485.436,E2 -4485.436} C_VEL
LIN {X 0,Y 531.037,Z 63.831,A -85,B 0,C 180,E1 -4488.549,E2 -4488.549} C_VEL
LIN {X 0,Y 531.055,Z 63.824,A -85,B 0,C 180,E1 -4491.629,E2 -4491.629} C_VEL
LIN {X 0,Y 531.121,Z 63.823,A -85,B 0,C 180,E1 -4494.685,E2 -4494.685} C_VEL
LIN {X 0,Y 531.141,Z 63.822,A -85,B 0,C 180,E1 -4497.725,E2 -4497.725} C_VEL
LIN {X 0,Y 531.152,Z 63.811,A -85,B 0,C 180,E1 -4500.758,E2 -4500.758} C_VEL
LIN {X 0,Y 531.103,Z 63.822,A -85,B 0,C 180,E1 -4503.034,E2 -4503.034} C_VEL
LIN {X 0,Y 531.084,Z 63.829,A -85,B 0,C 180,E1 -4506.077,E2 -4506.077} C_VEL
LIN {X 0,Y 531.028,Z 63.829,A -85,B 0,C 180,E1 -4509.138,E2 -4509.138} C_VEL
LIN {X 0,Y 531.04,Z 63.831,A -85,B 0,C 180,E1 -4512.225,E2 -4512.225} C_VEL
LIN {X 0,Y 530.995,Z 63.845,A -85,B 0,C 180,E1 -4515.349,E2 -4515.349} C_VEL
LIN {X 0,Y 530.989,Z 63.832,A -85,B 0,C 180,E1 -4518.521,E2 -4518.521} C_VEL
LIN {X 0,Y 530.999,Z 63.837,A -85,B 0,C 180,E1 -4520.937,E2 -4520.937} C_VEL
LIN {X 0,Y 530.978,Z 63.839,A -85,B 0,C 180,E1 -4524.224,E2 -4524.224} C_VEL
LIN {X 0,Y 531.003,Z 63.837,A -85,B 0,C 180,E1 -4526.743,E2 -4526.743} C_VEL
LIN {X 0,Y 530.98,Z 63.843,A -85,B 0,C 180,E1 -4529.322,E2 -4529.322} C_VEL
LIN {X 0,Y 530.978,Z 63.84,A -85,B 0,C 180,E1 -4532.103,E2 -4532.103} C_VEL
LIN {X 0,Y 530.987,Z 63.842,A -85,B 0,C 180,E1 -4534.854,E2 -4534.854} C_VEL
LIN {X 0,Y 530.964,Z 63.842,A -85,B 0,C 180,E1 -4537.507,E2 -4537.507} C_VEL
LIN {X 0,Y 530.998,Z 63.841,A -85,B 0,C 180,E1 -4540.431,E2 -4540.431} C_VEL
LIN {X 0,Y 530.961,Z 63.842,A -85,B 0,C 180,E1 -4543.494,E2 -4543.494} C_VEL
LIN {X 0,Y 530.959,Z 63.842,A -85,B 0,C 180,E1 -4543.561,E2 -4543.561} C_VEL
LIN {X 0,Y 530.285,Z 63.932,A -85,B 0,C 180,E1 -4544.194,E2 -4544.194} C_VEL
LIN {X 0,Y 527.435,Z 64.281,A -85,B 0,C 180,E1 -4545.223,E2 -4545.223} C_VEL
LIN {X 0,Y 525.031,Z 64.581,A -85,B 0,C 180,E1 -4546.052,E2 -4546.052} C_VEL
LIN {X 0,Y 523.998,Z 64.702,A -85,B 0,C 180,E1 -4546.691,E2 -4546.691} C_VEL
LIN {X 0,Y 523.914,Z 64.71,A -85,B 0,C 180,E1 -4546.908,E2 -4546.908} C_VEL
LIN {X 0,Y 523.942,Z 64.712,A -85,B 0,C 180,E1 -4548.908,E2 -4548.908} C_VEL
LIN {X 0,Y 523.914,Z 64.724,A -85,B 0,C 180,E1 -4551.898,E2 -4551.898} C_VEL
LIN {X 0,Y 523.936,Z 64.709,A -85,B 0,C 180,E1 -4554.909,E2 -4554.909} C_VEL
LIN {X 0,Y 523.935,Z 64.72,A -85,B 0,C 180,E1 -4557.679,E2 -4557.679} C_VEL
LIN {X 0,Y 523.951,Z 64.711,A -85,B 0,C 180,E1 -4560.676,E2 -4560.676} C_VEL
LIN {X 0,Y 523.972,Z 64.72,A -85,B 0,C 180,E1 -4563.729,E2 -4563.729} C_VEL
LIN {X 0,Y 523.933,Z 64.721,A -85,B 0,C 180,E1 -4566.271,E2 -4566.271} C_VEL
LIN {X 0,Y 523.943,Z 64.717,A -85,B 0,C 180,E1 -4568.767,E2 -4568.767} C_VEL
LIN {X 0,Y 523.949,Z 64.72,A -85,B 0,C 180,E1 -4571.221,E2 -4571.221} C_VEL
LIN {X 0,Y 523.935,Z 64.725,A -85,B 0,C 180,E1 -4573.639,E2 -4573.639} C_VEL
LIN {X 0,Y 523.942,Z 64.719,A -85,B 0,C 180,E1 -4576.028,E2 -4576.028} C_VEL
LIN {X 0,Y 524.009,Z 64.71,A -85,B 0,C 180,E1 -4578.394,E2 -4578.394} C_VEL
LIN {X 0,Y 524.002,Z 64.716,A -85,B 0,C 180,E1 -4581.516,E2 -4581.516} C_VEL
LIN {X 0,Y 524.084,Z 64.702,A -85,B 0,C 180,E1 -4584.614,E2 -4584.614} C_VEL
LIN {X 0,Y 524.111,Z 64.698,A -85,B 0,C 180,E1 -4587.694,E2 -4587.694} C_VEL
LIN {X 0,Y 524.121,Z 64.701,A -85,B 0,C 180,E1 -4590.768,E2 -4590.768} C_VEL
LIN {X 0,Y 524.069,Z 64.708,A -85,B 0,C 180,E1 -4593.075,E2 -4593.075} C_VEL
LIN {X 0,Y 524.05,Z 64.706,A -85,B 0,C 180,E1 -4596.159,E2 -4596.159} C_VEL
LIN {X 0,Y 523.997,Z 64.713,A -85,B 0,C 180,E1 -4599.262,E2 -4599.262} C_VEL
LIN {X 0,Y 524,Z 64.711,A -85,B 0,C 180,E1 -4601.74,E2 -4601.74} C_VEL
LIN {X 0,Y 523.991,Z 64.714,A -85,B 0,C 180,E1 -4605.053,E2 -4605.053} C_VEL
LIN {X 0,Y 523.961,Z 64.718,A -85,B 0,C 180,E1 -4607.969,E2 -4607.969} C_VEL
LIN {X 0,Y 523.969,Z 64.721,A -85,B 0,C 180,E1 -4610.41,E2 -4610.41} C_VEL
LIN {X 0,Y 523.914,Z 64.722,A -85,B 0,C 180,E1 -4612.893,E2 -4612.893} C_VEL
LIN {X 0,Y 523.95,Z 64.717,A -85,B 0,C 180,E1 -4615.419,E2 -4615.419} C_VEL
LIN {X 0,Y 523.967,Z 64.719,A -85,B 0,C 180,E1 -4617.999,E2 -4617.999} C_VEL
LIN {X 0,Y 523.944,Z 64.716,A -85,B 0,C 180,E1 -4620.855,E2 -4620.855} C_VEL
LIN {X 0,Y 523.958,Z 64.715,A -85,B 0,C 180,E1 -4623.735,E2 -4623.735} C_VEL
LIN {X 0,Y 523.92,Z 64.72,A -85,B 0,C 180,E1 -4626.405,E2 -4626.405} C_VEL
LIN {X 0,Y 523.92,Z 64.72,A -85,B 0,C 180,E1 -4629.085,E2 -4629.085} C_VEL
LIN {X 0,Y 523.949,Z 64.705,A -85,B 0,C 180,E1 -4632.119,E2 -4632.119} C_VEL
LIN {X 0,Y 523.952,Z 64.717,A -85,B 0,C 180,E1 -4635.309,E2 -4635.309} C_VEL
LIN {X 0,Y 523.969,Z 64.711,A -85,B 0,C 180,E1 -4638.688,E2 -4638.688} C_VEL
LIN {X 0,Y 523.917,Z 64.722,A -85,B 0,C 180,E1 -4641.08,E2 -4641.08} C_VEL
LIN {X 0,Y 523.926,Z 64.718,A -85,B 0,C 180,E1 -4643.828,E2 -4643.828} C_VEL
LIN {X 0,Y 523.94,Z 64.714,A -85,B 0,C 180,E1 -4646.636,E2 -4646.636} C_VEL
LIN {X 0,Y 523.954,Z 64.719,A -85,B 0,C 180,E1 -4649.356,E2 -4649.356} C_VEL
LIN {X 0,Y 523.977,Z 64.708,A -85,B 0,C 180,E1 -4652.281,E2 -4652.281} C_VEL
LIN {X 0,Y 523.951,Z 64.715,A -85,B 0,C 180,E1 -4654.582,E2 -4654.582} C_VEL
LIN {X 0,Y 523.915,Z 64.723,A -85,B 0,C 180,E1 -4657.107,E2 -4657.107} C_VEL
LIN {X 0,Y 523.977,Z 64.707,A -85,B 0,C 180,E1 -4659.866,E2 -4659.866} C_VEL
LIN {X 0,Y 523.966,Z 64.717,A -85,B 0,C 180,E1 -4662.838,E2 -4662.838} C_VEL
LIN {X 0,Y 523.976,Z 64.713,A -85,B 0,C 180,E1 -4665.236,E2 -4665.236} C_VEL
LIN {X 0,Y 524.014,Z 64.709,A -85,B 0,C 180,E1 -4668.395,E2 -4668.395} C_VEL
LIN {X 0,Y 524.003,Z 64.702,A -85,B 0,C 180,E1 -4671.516,E2 -4671.516} C_VEL
LIN {X 0,Y 524.082,Z 64.702,A -85,B 0,C 180,E1 -4674.614,E2 -4674.614} C_VEL
LIN {X 0,Y 524.112,Z 64.696,A -85,B 0,C 180,E1 -4677.695,E2 -4677.695} C_VEL
LIN {X 0,Y 524.123,Z 64.687,A -85,B 0,C 180,E1 -4680.769,E2 -4680.769} C_VEL
LIN {X 0,Y 524.07,Z 64.698,A -85,B 0,C 180,E1 -4683.075,E2 -4683.075} C_VEL
LIN {X 0,Y 524.047,Z 64.705,A -85,B 0,C 180,E1 -4686.159,E2 -4686.159} C_VEL
LIN {X 0,Y 523.997,Z 64.704,A -85,B 0,C 180,E1 -4689.262,E2 -4689.262} C_VEL
LIN {X 0,Y 524.004,Z 64.712,A -85,B 0,C 180,E1 -4691.74,E2 -4691.74} C_VEL
LIN {X 0,Y 523.994,Z 64.711,A -85,B 0,C 180,E1 -4695.053,E2 -4695.053} C_VEL
LIN {X 0,Y 523.965,Z 64.706,A -85,B 0,C 180,E1 -4697.969,E2 -4697.969} C_VEL
LIN {X 0,Y 523.973,Z 64.708,A -85,B 0,C 180,E1 -4700.41,E2 -4700.41} C_VEL
LIN {X 0,Y 523.918,Z 64.721,A -85,B 0,C 180,E1 -4702.894,E2 -4702.894} C_VEL
LIN {X 0,Y 523.954,Z 64.715,A -85,B 0,C 180,E1 -4705.419,E2 -4705.419} C_VEL
LIN {X 0,Y 523.969,Z 64.709,A -85,B 0,C 180,E1 -4707.999,E2 -4707.999} C_VEL
LIN {X 0,Y 523.946,Z 64.722,A -85,B 0,C 180,E1 -4710.855,E2 -4710.855} C_VEL
LIN {X 0,Y 523.962,Z 64.708,A -85,B 0,C 180,E1 -4713.735,E2 -4713.735} C_VEL
LIN {X 0,Y 523.905,Z 64.722,A -85,B 0,C 180,E1 -4716.402,E2 -4716.402} C_VEL
LIN {X 0,Y 523.924,Z 64.719,A -85,B 0,C 180,E1 -4719.085,E2 -4719.085} C_VEL
LIN {X 0,Y 523.953,Z 64.716,A -85,B 0,C 180,E1 -4722.119,E2 -4722.119} C_VEL
LIN {X 0,Y 523.943,Z 64.715,A -85,B 0,C 180,E1 -4725.311,E2 -4725.311} C_VEL
LIN {X 0,Y 523.957,Z 64.713,A -85,B 0,C 180,E1 -4728.69,E2 -4728.69} C_VEL
LIN {X 0,Y 523.918,Z 64.719,A -85,B 0,C 180,E1 -4731.081,E2 -4731.081} C_VEL
LIN {X 0,Y 523.925,Z 64.721,A -85,B 0,C 180,E1 -4733.827,E2 -4733.827} C_VEL
LIN {X 0,Y 523.944,Z 64.719,A -85,B 0,C 180,E1 -4736.636,E2 -4736.636} C_VEL
LIN {X 0,Y 523.958,Z 64.717,A -85,B 0,C 180,E1 -4739.356,E2 -4739.356} C_VEL
LIN {X 0,Y 523.982,Z 64.716,A -85,B 0,C 180,E1 -4742.281,E2 -4742.281} C_VEL
LIN {X 0,Y 523.994,Z 64.747,A -85,B 0,C 180,E1 -4743.979,E2 -4743.979} C_VEL
LIN {X 0,Y 525.082,Z 71.723,A -85,B 0,C 180,E1 -4745.527,E2 -4745.527} C_VEL
LIN {X 0,Y 524.717,Z 85.968,A -85,B 0,C 180,E1 -4748.387,E2 -4748.387} C_VEL
LIN {X 0,Y 524.4,Z 99.563,A -85,B 0,C 180,E1 -4751.035,E2 -4751.035} C_VEL
LIN {X 0,Y 524.167,Z 114.039,A -85,B 0,C 180,E1 -4753.846,E2 -4753.846} C_VEL
LIN {X 0,Y 524.023,Z 119.205,A -85,B 0,C 180,E1 -4754.827,E2 -4754.827} C_VEL
LIN {X 0,Y 525.204,Z 126.702,A -85,B 0,C 180,E1 -4754.996,E2 -4754.996} C_VEL
LIN {X 0,Y 525.9,Z 131.584,A -85,B 0,C 180,E1 -4755.083,E2 -4755.083} C_VEL
LIN {X 0,Y 525.527,Z 224.047,A -85,B 0,C 180,E1 -4756.367,E2 -4756.367} C_VEL
LIN {X 0,Y 525.316,Z 234.818,A -85,B 0,C 180,E1 -4756.608,E2 -4756.608} C_VEL
LIN {X 0,Y 525.197,Z 243.923,A -85,B 0,C 180,E1 -4756.9,E2 -4756.9} C_VEL
LIN {X 0,Y 524.999,Z 253.282,A -85,B 0,C 180,E1 -4757.288,E2 -4757.288} C_VEL
LIN {X 0,Y 524.757,Z 263.414,A -85,B 0,C 180,E1 -4757.822,E2 -4757.822} C_VEL
LIN {X 0,Y 524.513,Z 272.427,A -85,B 0,C 180,E1 -4758.405,E2 -4758.405} C_VEL
LIN {X 0,Y 524.328,Z 281.159,A -85,B 0,C 180,E1 -4759.086,E2 -4759.086} C_VEL
LIN {X 0,Y 524.132,Z 288.556,A -85,B 0,C 180,E1 -4759.766,E2 -4759.766} C_VEL
LIN {X 0,Y 523.945,Z 295.777,A -85,B 0,C 180,E1 -4760.542,E2 -4760.542} C_VEL
LIN {X 0,Y 523.779,Z 301.979,A -85,B 0,C 180,E1 -4761.318,E2 -4761.318} C_VEL
LIN {X 0,Y 523.622,Z 308.516,A -85,B 0,C 180,E1 -4762.287,E2 -4762.287} C_VEL
LIN {X 0,Y 523.493,Z 314.018,A -85,B 0,C 180,E1 -4763.263,E2 -4763.263} C_VEL
LIN {X 0,Y 523.479,Z 318.505,A -85,B 0,C 180,E1 -4764.221,E2 -4764.221} C_VEL
LIN {X 0,Y 523.359,Z 322.823,A -85,B 0,C 180,E1 -4765.379,E2 -4765.379} C_VEL
LIN {X 0,Y 523.443,Z 325.189,A -85,B 0,C 180,E1 -4766.151,E2 -4766.151} C_VEL
LIN {X 0,Y 523.368,Z 326.982,A -85,B 0,C 180,E1 -4766.921,E2 -4766.921} C_VEL
LIN {X 0,Y 523.275,Z 329.419,A -85,B 0,C 180,E1 -4768.461,E2 -4768.461} C_VEL
LIN {X 0,Y 523.254,Z 330.005,A -85,B 0,C 180,E1 -4769.23,E2 -4769.23} C_VEL
LIN {X 0,Y 523.254,Z 330.005,A -85,B 0,C 180,E1 -4770.77,E2 -4770.77} C_VEL
LIN {X 0,Y 523.275,Z 329.419,A -85,B 0,C 180,E1 -4771.539,E2 -4771.539} C_VEL
LIN {X 0,Y 523.368,Z 326.982,A -85,B 0,C 180,E1 -4773.079,E2 -4773.079} C_VEL
LIN {X 0,Y 523.424,Z 324.04,A -85,B 0,C 180,E1 -4774.235,E2 -4774.235} C_VEL
LIN {X 0,Y 523.452,Z 320.057,A -85,B 0,C 180,E1 -4775.393,E2 -4775.393} C_VEL
LIN {X 0,Y 523.467,Z 315.06,A -85,B 0,C 180,E1 -4776.527,E2 -4776.527} C_VEL
LIN {X 0,Y 523.59,Z 309.671,A -85,B 0,C 180,E1 -4777.52,E2 -4777.52} C_VEL
LIN {X 0,Y 523.751,Z 303.356,A -85,B 0,C 180,E1 -4778.488,E2 -4778.488} C_VEL
LIN {X 0,Y 523.883,Z 297.404,A -85,B 0,C 180,E1 -4779.264,E2 -4779.264} C_VEL
LIN {X 0,Y 524.019,Z 290.474,A -85,B 0,C 180,E1 -4780.041,E2 -4780.041} C_VEL
LIN {X 0,Y 524.309,Z 282.294,A -85,B 0,C 180,E1 -4780.816,E2 -4780.816} C_VEL
LIN {X 0,Y 524.521,Z 273.78,A -85,B 0,C 180,E1 -4781.496,E2 -4781.496} C_VEL
LIN {X 0,Y 524.702,Z 264.746,A -85,B 0,C 180,E1 -4782.099,E2 -4782.099} C_VEL
LIN {X 0,Y 524.975,Z 255.298,A -85,B 0,C 180,E1 -4782.614,E2 -4782.614} C_VEL
LIN {X 0,Y 525.162,Z 246.5,A -85,B 0,C 180,E1 -4783.002,E2 -4783.002} C_VEL
LIN {X 0,Y 525.327,Z 236.568,A -85,B 0,C 180,E1 -4783.343,E2 -4783.343} C_VEL
LIN {X 0,Y 525.469,Z 226.71,A -85,B 0,C 180,E1 -4783.585,E2 -4783.585} C_VEL
LIN {X 0,Y 525.681,Z 202.1,A -85,B 0,C 180,E1 -4783.949,E2 -4783.949} C_VEL
LIN {X 0,Y 525.759,Z 129.887,A -85,B 0,C 180,E1 -4784.944,E2 -4784.944} C_VEL
LIN {X 0,Y 524.069,Z 119.617,A -85,B 0,C 180,E1 -4785.147,E2 -4785.147} C_VEL
LIN {X 0,Y 524.024,Z 118.459,A -85,B 0,C 180,E1 -4785.28,E2 -4785.28} C_VEL
LIN {X 0,Y 524.285,Z 107.037,A -85,B 0,C 180,E1 -4787.523,E2 -4787.523} C_VEL
LIN {X 0,Y 524.601,Z 91.199,A -85,B 0,C 180,E1 -4790.589,E2 -4790.589} C_VEL
LIN {X 0,Y 525.031,Z 75.664,A -85,B 0,C 180,E1 -4793.677,E2 -4793.677} C_VEL
LIN {X 0,Y 525.005,Z 70.521,A -85,B 0,C 180,E1 -4794.729,E2 -4794.729} C_VEL
LIN {X 0,Y 523.993,Z 64.746,A -85,B 0,C 180,E1 -4796.021,E2 -4796.021} C_VEL
LIN {X 0,Y 523.942,Z 64.719,A -85,B 0,C 180,E1 -4798.874,E2 -4798.874} C_VEL
LIN {X 0,Y 523.923,Z 64.725,A -85,B 0,C 180,E1 -4801.544,E2 -4801.544} C_VEL
LIN {X 0,Y 523.944,Z 64.717,A -85,B 0,C 180,E1 -4804.289,E2 -4804.289} C_VEL
LIN {X 0,Y 523.912,Z 64.722,A -85,B 0,C 180,E1 -4807.132,E2 -4807.132} C_VEL
LIN {X 0,Y 523.94,Z 64.712,A -85,B 0,C 180,E1 -4810.13,E2 -4810.13} C_VEL
LIN {X 0,Y 523.937,Z 64.717,A -85,B 0,C 180,E1 -4812.459,E2 -4812.459} C_VEL
LIN {X 0,Y 523.943,Z 64.721,A -85,B 0,C 180,E1 -4815.31,E2 -4815.31} C_VEL
LIN {X 0,Y 523.957,Z 64.715,A -85,B 0,C 180,E1 -4818.689,E2 -4818.689} C_VEL
LIN {X 0,Y 523.921,Z 64.722,A -85,B 0,C 180,E1 -4821.08,E2 -4821.08} C_VEL
LIN {X 0,Y 523.903,Z 64.72,A -85,B 0,C 180,E1 -4823.825,E2 -4823.825} C_VEL
LIN {X 0,Y 523.943,Z 64.713,A -85,B 0,C 180,E1 -4826.635,E2 -4826.635} C_VEL
LIN {X 0,Y 523.957,Z 64.717,A -85,B 0,C 180,E1 -4829.355,E2 -4829.355} C_VEL
LIN {X 0,Y 523.978,Z 64.709,A -85,B 0,C 180,E1 -4832.281,E2 -4832.281} C_VEL
LIN {X 0,Y 523.954,Z 64.715,A -85,B 0,C 180,E1 -4834.581,E2 -4834.581} C_VEL
LIN {X 0,Y 523.918,Z 64.721,A -85,B 0,C 180,E1 -4837.106,E2 -4837.106} C_VEL
LIN {X 0,Y 523.98,Z 64.707,A -85,B 0,C 180,E1 -4839.866,E2 -4839.866} C_VEL
LIN {X 0,Y 523.967,Z 64.714,A -85,B 0,C 180,E1 -4842.837,E2 -4842.837} C_VEL
LIN {X 0,Y 523.978,Z 64.711,A -85,B 0,C 180,E1 -4845.235,E2 -4845.235} C_VEL
LIN {X 0,Y 524.013,Z 64.708,A -85,B 0,C 180,E1 -4848.394,E2 -4848.394} C_VEL
LIN {X 0,Y 524.004,Z 64.702,A -85,B 0,C 180,E1 -4851.516,E2 -4851.516} C_VEL
LIN {X 0,Y 524.082,Z 64.701,A -85,B 0,C 180,E1 -4854.613,E2 -4854.613} C_VEL
LIN {X 0,Y 524.113,Z 64.697,A -85,B 0,C 180,E1 -4857.694,E2 -4857.694} C_VEL
LIN {X 0,Y 524.123,Z 64.686,A -85,B 0,C 180,E1 -4860.768,E2 -4860.768} C_VEL
LIN {X 0,Y 524.07,Z 64.698,A -85,B 0,C 180,E1 -4863.074,E2 -4863.074} C_VEL
LIN {X 0,Y 524.046,Z 64.705,A -85,B 0,C 180,E1 -4866.159,E2 -4866.159} C_VEL
LIN {X 0,Y 523.996,Z 64.706,A -85,B 0,C 180,E1 -4869.261,E2 -4869.261} C_VEL
LIN {X 0,Y 524.024,Z 64.71,A -85,B 0,C 180,E1 -4871.751,E2 -4871.751} C_VEL
LIN {X 0,Y 523.992,Z 64.713,A -85,B 0,C 180,E1 -4875.052,E2 -4875.052} C_VEL
LIN {X 0,Y 523.963,Z 64.708,A -85,B 0,C 180,E1 -4877.969,E2 -4877.969} C_VEL
LIN {X 0,Y 523.971,Z 64.708,A -85,B 0,C 180,E1 -4880.41,E2 -4880.41} C_VEL
LIN {X 0,Y 523.915,Z 64.723,A -85,B 0,C 180,E1 -4882.893,E2 -4882.893} C_VEL
LIN {X 0,Y 523.951,Z 64.715,A -85,B 0,C 180,E1 -4885.418,E2 -4885.418} C_VEL
LIN {X 0,Y 523.968,Z 64.708,A -85,B 0,C 180,E1 -4887.998,E2 -4887.998} C_VEL
LIN {X 0,Y 523.945,Z 64.723,A -85,B 0,C 180,E1 -4890.855,E2 -4890.855} C_VEL
LIN {X 0,Y 523.959,Z 64.71,A -85,B 0,C 180,E1 -4893.735,E2 -4893.735} C_VEL
LIN {X 0,Y 523.92,Z 64.721,A -85,B 0,C 180,E1 -4896.404,E2 -4896.404} C_VEL
LIN {X 0,Y 523.92,Z 64.72,A -85,B 0,C 180,E1 -4899.084,E2 -4899.084} C_VEL
LIN {X 0,Y 523.969,Z 64.711,A -85,B 0,C 180,E1 -4901.312,E2 -4901.312} C_VEL
LIN {X 0,Y 523.952,Z 64.717,A -85,B 0,C 180,E1 -4904.691,E2 -4904.691} C_VEL
LIN {X 0,Y 523.914,Z 64.71,A -85,B 0,C 180,E1 -4906.908,E2 -4906.908} C_VEL
LIN {X 0,Y 523.249,Z 64.791,A -85,B 0,C 180,E1 -4907.549,E2 -4907.549} C_VEL
LIN {X 0,Y 520.407,Z 65.151,A -85,B 0,C 180,E1 -4908.591,E2 -4908.591} C_VEL
LIN {X 0,Y 518.002,Z 65.457,A -85,B 0,C 180,E1 -4909.43,E2 -4909.43} C_VEL
LIN {X 0,Y 516.965,Z 65.588,A -85,B 0,C 180,E1 -4910.078,E2 -4910.078} C_VEL
LIN {X 0,Y 516.879,Z 65.598,A -85,B 0,C 180,E1 -4910.297,E2 -4910.297} C_VEL
LIN {X 0,Y 516.882,Z 65.595,A -85,B 0,C 180,E1 -4913.342,E2 -4913.342} C_VEL
LIN {X 0,Y 516.909,Z 65.59,A -85,B 0,C 180,E1 -4916.121,E2 -4916.121} C_VEL
LIN {X 0,Y 516.888,Z 65.595,A -85,B 0,C 180,E1 -4918.935,E2 -4918.935} C_VEL
LIN {X 0,Y 516.916,Z 65.59,A -85,B 0,C 180,E1 -4921.585,E2 -4921.585} C_VEL
LIN {X 0,Y 516.928,Z 65.595,A -85,B 0,C 180,E1 -4924.211,E2 -4924.211} C_VEL
LIN {X 0,Y 516.869,Z 65.599,A -85,B 0,C 180,E1 -4926.776,E2 -4926.776} C_VEL
LIN {X 0,Y 516.936,Z 65.597,A -85,B 0,C 180,E1 -4929.731,E2 -4929.731} C_VEL
LIN {X 0,Y 516.926,Z 65.592,A -85,B 0,C 180,E1 -4932.596,E2 -4932.596} C_VEL
LIN {X 0,Y 516.948,Z 65.592,A -85,B 0,C 180,E1 -4935.03,E2 -4935.03} C_VEL
LIN {X 0,Y 516.962,Z 65.588,A -85,B 0,C 180,E1 -4938.234,E2 -4938.234} C_VEL
LIN {X 0,Y 516.967,Z 65.593,A -85,B 0,C 180,E1 -4941.4,E2 -4941.4} C_VEL
LIN {X 0,Y 517.013,Z 65.583,A -85,B 0,C 180,E1 -4943.757,E2 -4943.757} C_VEL
LIN {X 0,Y 517.083,Z 65.574,A -85,B 0,C 180,E1 -4947.663,E2 -4947.663} C_VEL
LIN {X 0,Y 517.091,Z 65.577,A -85,B 0,C 180,E1 -4950.779,E2 -4950.779} C_VEL
LIN {X 0,Y 517.01,Z 65.587,A -85,B 0,C 180,E1 -4953.117,E2 -4953.117} C_VEL
LIN {X 0,Y 517.013,Z 65.583,A -85,B 0,C 180,E1 -4956.243,E2 -4956.243} C_VEL
LIN {X 0,Y 516.951,Z 65.59,A -85,B 0,C 180,E1 -4959.389,E2 -4959.389} C_VEL
LIN {X 0,Y 516.949,Z 65.59,A -85,B 0,C 180,E1 -4961.808,E2 -4961.808} C_VEL
LIN {X 0,Y 516.944,Z 65.591,A -85,B 0,C 180,E1 -4965.148,E2 -4965.148} C_VEL
LIN {X 0,Y 516.922,Z 65.598,A -85,B 0,C 180,E1 -4968.222,E2 -4968.222} C_VEL
LIN {X 0,Y 516.909,Z 65.597,A -85,B 0,C 180,E1 -4970.702,E2 -4970.702} C_VEL
LIN {X 0,Y 516.908,Z 65.6,A -85,B 0,C 180,E1 -4974.072,E2 -4974.072} C_VEL
LIN {X 0,Y 516.923,Z 65.594,A -85,B 0,C 180,E1 -4976.658,E2 -4976.658} C_VEL
LIN {X 0,Y 516.908,Z 65.589,A -85,B 0,C 180,E1 -4979.524,E2 -4979.524} C_VEL
LIN {X 0,Y 516.898,Z 65.594,A -85,B 0,C 180,E1 -4982.545,E2 -4982.545} C_VEL
LIN {X 0,Y 516.88,Z 65.586,A -85,B 0,C 180,E1 -4985.333,E2 -4985.333} C_VEL
LIN {X 0,Y 516.879,Z 65.602,A -85,B 0,C 180,E1 -4987.944,E2 -4987.944} C_VEL
LIN {X 0,Y 516.881,Z 65.589,A -85,B 0,C 180,E1 -4990.742,E2 -4990.742} C_VEL
LIN {X 0,Y 516.875,Z 65.584,A -85,B 0,C 180,E1 -4992.832,E2 -4992.832} C_VEL
LIN {X 0,Y 516.919,Z 65.59,A -85,B 0,C 180,E1 -4995.01,E2 -4995.01} C_VEL
LIN {X 0,Y 516.919,Z 65.589,A -85,B 0,C 180,E1 -4998.398,E2 -4998.398} C_VEL
LIN {X 0,Y 516.88,Z 65.602,A -85,B 0,C 180,E1 -5001.285,E2 -5001.285} C_VEL
LIN {X 0,Y 516.888,Z 65.593,A -85,B 0,C 180,E1 -5004.222,E2 -5004.222} C_VEL
LIN {X 0,Y 516.894,Z 65.597,A -85,B 0,C 180,E1 -5007.054,E2 -5007.054} C_VEL
LIN {X 0,Y 516.89,Z 65.595,A -85,B 0,C 180,E1 -5009.797,E2 -5009.797} C_VEL
LIN {X 0,Y 516.926,Z 65.587,A -85,B 0,C 180,E1 -5012.468,E2 -5012.468} C_VEL
LIN {X 0,Y 516.909,Z 65.598,A -85,B 0,C 180,E1 -5015.072,E2 -5015.072} C_VEL
LIN {X 0,Y 516.868,Z 65.597,A -85,B 0,C 180,E1 -5017.622,E2 -5017.622} C_VEL
LIN {X 0,Y 516.931,Z 65.586,A -85,B 0,C 180,E1 -5020.13,E2 -5020.13} C_VEL
LIN {X 0,Y 516.928,Z 65.591,A -85,B 0,C 180,E1 -5022.597,E2 -5022.597} C_VEL
LIN {X 0,Y 516.941,Z 65.59,A -85,B 0,C 180,E1 -5025.031,E2 -5025.031} C_VEL
LIN {X 0,Y 517.004,Z 65.584,A -85,B 0,C 180,E1 -5028.235,E2 -5028.235} C_VEL
LIN {X 0,Y 516.968,Z 65.578,A -85,B 0,C 180,E1 -5031.4,E2 -5031.4} C_VEL
LIN {X 0,Y 517.01,Z 65.58,A -85,B 0,C 180,E1 -5033.757,E2 -5033.757} C_VEL
LIN {X 0,Y 517.084,Z 65.571,A -85,B 0,C 180,E1 -5037.664,E2 -5037.664} C_VEL
LIN {X 0,Y 517.093,Z 65.562,A -85,B 0,C 180,E1 -5040.779,E2 -5040.779} C_VEL
LIN {X 0,Y 517.011,Z 65.578,A -85,B 0,C 180,E1 -5043.117,E2 -5043.117} C_VEL
LIN {X 0,Y 517.011,Z 65.581,A -85,B 0,C 180,E1 -5046.244,E2 -5046.244} C_VEL
LIN {X 0,Y 516.952,Z 65.583,A -85,B 0,C 180,E1 -5049.39,E2 -5049.39} C_VEL
LIN {X 0,Y 516.953,Z 65.591,A -85,B 0,C 180,E1 -5051.808,E2 -5051.808} C_VEL
LIN {X 0,Y 516.945,Z 65.59,A -85,B 0,C 180,E1 -5055.147,E2 -5055.147} C_VEL
LIN {X 0,Y 516.926,Z 65.581,A -85,B 0,C 180,E1 -5058.223,E2 -5058.223} C_VEL
LIN {X 0,Y 516.914,Z 65.588,A -85,B 0,C 180,E1 -5060.702,E2 -5060.702} C_VEL
LIN {X 0,Y 516.913,Z 65.591,A -85,B 0,C 180,E1 -5064.072,E2 -5064.072} C_VEL
LIN {X 0,Y 516.925,Z 65.586,A -85,B 0,C 180,E1 -5066.658,E2 -5066.658} C_VEL
LIN {X 0,Y 516.912,Z 65.594,A -85,B 0,C 180,E1 -5069.524,E2 -5069.524} C_VEL
LIN {X 0,Y 516.897,Z 65.596,A -85,B 0,C 180,E1 -5072.544,E2 -5072.544} C_VEL
LIN {X 0,Y 516.871,Z 65.598,A -85,B 0,C 180,E1 -5075.331,E2 -5075.331} C_VEL
LIN {X 0,Y 516.882,Z 65.596,A -85,B 0,C 180,E1 -5077.944,E2 -5077.944} C_VEL
LIN {X 0,Y 516.884,Z 65.599,A -85,B 0,C 180,E1 -5080.742,E2 -5080.742} C_VEL
LIN {X 0,Y 516.884,Z 65.601,A -85,B 0,C 180,E1 -5082.832,E2 -5082.832} C_VEL
LIN {X 0,Y 516.897,Z 65.596,A -85,B 0,C 180,E1 -5085.007,E2 -5085.007} C_VEL
LIN {X 0,Y 516.915,Z 65.595,A -85,B 0,C 180,E1 -5088.399,E2 -5088.399} C_VEL
LIN {X 0,Y 516.881,Z 65.595,A -85,B 0,C 180,E1 -5091.284,E2 -5091.284} C_VEL
LIN {X 0,Y 516.889,Z 65.597,A -85,B 0,C 180,E1 -5094.221,E2 -5094.221} C_VEL
LIN {X 0,Y 516.897,Z 65.594,A -85,B 0,C 180,E1 -5097.053,E2 -5097.053} C_VEL
LIN {X 0,Y 516.895,Z 65.601,A -85,B 0,C 180,E1 -5099.797,E2 -5099.797} C_VEL
LIN {X 0,Y 516.931,Z 65.594,A -85,B 0,C 180,E1 -5102.468,E2 -5102.468} C_VEL
LIN {X 0,Y 516.951,Z 65.624,A -85,B 0,C 180,E1 -5103.803,E2 -5103.803} C_VEL
LIN {X 0,Y 518.099,Z 72.454,A -85,B 0,C 180,E1 -5105.348,E2 -5105.348} C_VEL
LIN {X 0,Y 517.803,Z 83.767,A -85,B 0,C 180,E1 -5107.664,E2 -5107.664} C_VEL
LIN {X 0,Y 517.467,Z 98.388,A -85,B 0,C 180,E1 -5110.564,E2 -5110.564} C_VEL
LIN {X 0,Y 517.158,Z 113.879,A -85,B 0,C 180,E1 -5113.621,E2 -5113.621} C_VEL
LIN {X 0,Y 517.003,Z 119.099,A -85,B 0,C 180,E1 -5114.622,E2 -5114.622} C_VEL
LIN {X 0,Y 519.035,Z 132.685,A -85,B 0,C 180,E1 -5114.899,E2 -5114.899} C_VEL
LIN {X 0,Y 518.644,Z 223.857,A -85,B 0,C 180,E1 -5116.182,E2 -5116.182} C_VEL
LIN {X 0,Y 518.407,Z 234.628,A -85,B 0,C 180,E1 -5116.426,E2 -5116.426} C_VEL
LIN {X 0,Y 518.29,Z 243.733,A -85,B 0,C 180,E1 -5116.722,E2 -5116.722} C_VEL
LIN {X 0,Y 518.056,Z 253.091,A -85,B 0,C 180,E1 -5117.115,E2 -5117.115} C_VEL
LIN {X 0,Y 517.801,Z 263.326,A -85,B 0,C 180,E1 -5117.662,E2 -5117.662} C_VEL
LIN {X 0,Y 517.532,Z 272.235,A -85,B 0,C 180,E1 -5118.247,E2 -5118.247} C_VEL
LIN {X 0,Y 517.328,Z 280.968,A -85,B 0,C 180,E1 -5118.937,E2 -5118.937} C_VEL
LIN {X 0,Y 517.106,Z 288.365,A -85,B 0,C 180,E1 -5119.626,E2 -5119.626} C_VEL
LIN {X 0,Y 516.919,Z 295.586,A -85,B 0,C 180,E1 -5120.413,E2 -5120.413} C_VEL
LIN {X 0,Y 516.701,Z 301.787,A -85,B 0,C 180,E1 -5121.198,E2 -5121.198} C_VEL
LIN {X 0,Y 516.543,Z 308.324,A -85,B 0,C 180,E1 -5122.18,E2 -5122.18} C_VEL
LIN {X 0,Y 516.436,Z 312.824,A -85,B 0,C 180,E1 -5122.965,E2 -5122.965} C_VEL
LIN {X 0,Y 516.393,Z 318.314,A -85,B 0,C 180,E1 -5124.141,E2 -5124.141} C_VEL
LIN {X 0,Y 516.271,Z 322.632,A -85,B 0,C 180,E1 -5125.315,E2 -5125.315} C_VEL
LIN {X 0,Y 516.352,Z 324.998,A -85,B 0,C 180,E1 -5126.098,E2 -5126.098} C_VEL
LIN {X 0,Y 516.283,Z 326.792,A -85,B 0,C 180,E1 -5126.879,E2 -5126.879} C_VEL
LIN {X 0,Y 516.192,Z 329.229,A -85,B 0,C 180,E1 -5128.44,E2 -5128.44} C_VEL
LIN {X 0,Y 516.164,Z 329.815,A -85,B 0,C 180,E1 -5129.22,E2 -5129.22} C_VEL
LIN {X 0,Y 516.164,Z 329.815,A -85,B 0,C 180,E1 -5130.78,E2 -5130.78} C_VEL
LIN {X 0,Y 516.192,Z 329.229,A -85,B 0,C 180,E1 -5131.56,E2 -5131.56} C_VEL
LIN {X 0,Y 516.283,Z 326.792,A -85,B 0,C 180,E1 -5133.121,E2 -5133.121} C_VEL
LIN {X 0,Y 516.312,Z 323.849,A -85,B 0,C 180,E1 -5134.293,E2 -5134.293} C_VEL
LIN {X 0,Y 516.364,Z 319.866,A -85,B 0,C 180,E1 -5135.467,E2 -5135.467} C_VEL
LIN {X 0,Y 516.382,Z 314.708,A -85,B 0,C 180,E1 -5136.649,E2 -5136.649} C_VEL
LIN {X 0,Y 516.528,Z 309.48,A -85,B 0,C 180,E1 -5137.623,E2 -5137.623} C_VEL
LIN {X 0,Y 516.704,Z 303.164,A -85,B 0,C 180,E1 -5138.605,E2 -5138.605} C_VEL
LIN {X 0,Y 516.844,Z 297.212,A -85,B 0,C 180,E1 -5139.391,E2 -5139.391} C_VEL
LIN {X 0,Y 517.006,Z 290.283,A -85,B 0,C 180,E1 -5140.179,E2 -5140.179} C_VEL
LIN {X 0,Y 517.31,Z 282.103,A -85,B 0,C 180,E1 -5140.964,E2 -5140.964} C_VEL
LIN {X 0,Y 517.541,Z 273.589,A -85,B 0,C 180,E1 -5141.654,E2 -5141.654} C_VEL
LIN {X 0,Y 517.715,Z 265.581,A -85,B 0,C 180,E1 -5142.203,E2 -5142.203} C_VEL
LIN {X 0,Y 518.013,Z 256.114,A -85,B 0,C 180,E1 -5142.736,E2 -5142.736} C_VEL
LIN {X 0,Y 518.236,Z 246.309,A -85,B 0,C 180,E1 -5143.179,E2 -5143.179} C_VEL
LIN {X 0,Y 518.405,Z 236.377,A -85,B 0,C 180,E1 -5143.524,E2 -5143.524} C_VEL
LIN {X 0,Y 518.575,Z 226.52,A -85,B 0,C 180,E1 -5143.769,E2 -5143.769} C_VEL
LIN {X 0,Y 518.796,Z 201.91,A -85,B 0,C 180,E1 -5144.138,E2 -5144.138} C_VEL
LIN {X 0,Y 518.86,Z 130.347,A -85,B 0,C 180,E1 -5145.139,E2 -5145.139} C_VEL
LIN {X 0,Y 517.036,Z 119.265,A -85,B 0,C 180,E1 -5145.366,E2 -5145.366} C_VEL
LIN {X 0,Y 517.017,Z 118.015,A -85,B 0,C 180,E1 -5145.547,E2 -5145.547} C_VEL
LIN {X 0,Y 517.388,Z 103.614,A -85,B 0,C 180,E1 -5148.41,E2 -5148.41} C_VEL
LIN {X 0,Y 517.668,Z 88.976,A -85,B 0,C 180,E1 -5151.295,E2 -5151.295} C_VEL
LIN {X 0,Y 518.118,Z 75.566,A -85,B 0,C 180,E1 -5154.012,E2 -5154.012} C_VEL
LIN {X 0,Y 517.844,Z 70.417,A -85,B 0,C 180,E1 -5155.095,E2 -5155.095} C_VEL
LIN {X 0,Y 516.95,Z 65.618,A -85,B 0,C 180,E1 -5156.197,E2 -5156.197} C_VEL
LIN {X 0,Y 516.924,Z 65.594,A -85,B 0,C 180,E1 -5159.304,E2 -5159.304} C_VEL
LIN {X 0,Y 516.898,Z 65.595,A -85,B 0,C 180,E1 -5162.543,E2 -5162.543} C_VEL
LIN {X 0,Y 516.882,Z 65.597,A -85,B 0,C 180,E1 -5165.331,E2 -5165.331} C_VEL
LIN {X 0,Y 516.882,Z 65.599,A -85,B 0,C 180,E1 -5167.943,E2 -5167.943} C_VEL
LIN {X 0,Y 516.885,Z 65.589,A -85,B 0,C 180,E1 -5170.741,E2 -5170.741} C_VEL
LIN {X 0,Y 516.884,Z 65.596,A -85,B 0,C 180,E1 -5172.831,E2 -5172.831} C_VEL
LIN {X 0,Y 516.897,Z 65.596,A -85,B 0,C 180,E1 -5175.007,E2 -5175.007} C_VEL
LIN {X 0,Y 516.915,Z 65.591,A -85,B 0,C 180,E1 -5178.398,E2 -5178.398} C_VEL
LIN {X 0,Y 516.884,Z 65.602,A -85,B 0,C 180,E1 -5181.284,E2 -5181.284} C_VEL
LIN {X 0,Y 516.874,Z 65.595,A -85,B 0,C 180,E1 -5184.22,E2 -5184.22} C_VEL
LIN {X 0,Y 516.896,Z 65.597,A -85,B 0,C 180,E1 -5187.053,E2 -5187.053} C_VEL
LIN {X 0,Y 516.893,Z 65.594,A -85,B 0,C 180,E1 -5189.796,E2 -5189.796} C_VEL
LIN {X 0,Y 516.927,Z 65.589,A -85,B 0,C 180,E1 -5192.467,E2 -5192.467} C_VEL
LIN {X 0,Y 516.912,Z 65.595,A -85,B 0,C 180,E1 -5195.072,E2 -5195.072} C_VEL
LIN {X 0,Y 516.871,Z 65.596,A -85,B 0,C 180,E1 -5197.621,E2 -5197.621} C_VEL
LIN {X 0,Y 516.933,Z 65.587,A -85,B 0,C 180,E1 -5200.129,E2 -5200.129} C_VEL
LIN {X 0,Y 516.922,Z 65.591,A -85,B 0,C 180,E1 -5202.596,E2 -5202.596} C_VEL
LIN {X 0,Y 516.943,Z 65.589,A -85,B 0,C 180,E1 -5205.03,E2 -5205.03} C_VEL
LIN {X 0,Y 516.966,Z 65.588,A -85,B 0,C 180,E1 -5208.233,E2 -5208.233} C_VEL
LIN {X 0,Y 516.969,Z 65.577,A -85,B 0,C 180,E1 -5211.399,E2 -5211.399} C_VEL
LIN {X 0,Y 517.011,Z 65.581,A -85,B 0,C 180,E1 -5213.756,E2 -5213.756} C_VEL
LIN {X 0,Y 517.085,Z 65.572,A -85,B 0,C 180,E1 -5217.663,E2 -5217.663} C_VEL
LIN {X 0,Y 517.093,Z 65.561,A -85,B 0,C 180,E1 -5220.778,E2 -5220.778} C_VEL
LIN {X 0,Y 517.011,Z 65.578,A -85,B 0,C 180,E1 -5223.117,E2 -5223.117} C_VEL
LIN {X 0,Y 517.01,Z 65.58,A -85,B 0,C 180,E1 -5226.243,E2 -5226.243} C_VEL
LIN {X 0,Y 516.951,Z 65.585,A -85,B 0,C 180,E1 -5229.389,E2 -5229.389} C_VEL
LIN {X 0,Y 516.983,Z 65.586,A -85,B 0,C 180,E1 -5231.824,E2 -5231.824} C_VEL
LIN {X 0,Y 516.943,Z 65.592,A -85,B 0,C 180,E1 -5235.146,E2 -5235.146} C_VEL
LIN {X 0,Y 516.924,Z 65.583,A -85,B 0,C 180,E1 -5238.222,E2 -5238.222} C_VEL
LIN {X 0,Y 516.911,Z 65.588,A -85,B 0,C 180,E1 -5240.701,E2 -5240.701} C_VEL
LIN {X 0,Y 516.91,Z 65.592,A -85,B 0,C 180,E1 -5244.072,E2 -5244.072} C_VEL
LIN {X 0,Y 516.924,Z 65.589,A -85,B 0,C 180,E1 -5246.657,E2 -5246.657} C_VEL
LIN {X 0,Y 516.909,Z 65.594,A -85,B 0,C 180,E1 -5249.523,E2 -5249.523} C_VEL
LIN {X 0,Y 516.898,Z 65.597,A -85,B 0,C 180,E1 -5252.544,E2 -5252.544} C_VEL
LIN {X 0,Y 516.881,Z 65.596,A -85,B 0,C 180,E1 -5255.332,E2 -5255.332} C_VEL
LIN {X 0,Y 516.879,Z 65.597,A -85,B 0,C 180,E1 -5257.943,E2 -5257.943} C_VEL
LIN {X 0,Y 516.901,Z 65.596,A -85,B 0,C 180,E1 -5260.739,E2 -5260.739} C_VEL
LIN {X 0,Y 516.879,Z 65.597,A -85,B 0,C 180,E1 -5263.903,E2 -5263.903} C_VEL
LIN {X 0,Y 516.879,Z 65.597,A -85,B 0,C 180,E1 -5266.107,E2 -5266.107} C_VEL
LIN {X 0,Y 516.914,Z 65.584,A -85,B 0,C 180,E1 -5268.398,E2 -5268.398} C_VEL
LIN {X 0,Y 516.879,Z 65.598,A -85,B 0,C 180,E1 -5270.297,E2 -5270.297} C_VEL
LIN {X 0,Y 516.209,Z 65.682,A -85,B 0,C 180,E1 -5270.947,E2 -5270.947} C_VEL
LIN {X 0,Y 513.364,Z 66.04,A -85,B 0,C 180,E1 -5272.003,E2 -5272.003} C_VEL
LIN {X 0,Y 510.957,Z 66.34,A -85,B 0,C 180,E1 -5272.853,E2 -5272.853} C_VEL
LIN {X 0,Y 509.917,Z 66.466,A -85,B 0,C 180,E1 -5273.509,E2 -5273.509} C_VEL
LIN {X 0,Y 509.829,Z 66.474,A -85,B 0,C 180,E1 -5273.732,E2 -5273.732} C_VEL
LIN {X 0,Y 509.859,Z 66.472,A -85,B 0,C 180,E1 -5276.539,E2 -5276.539} C_VEL
LIN {X 0,Y 509.842,Z 66.474,A -85,B 0,C 180,E1 -5279.334,E2 -5279.334} C_VEL
LIN {X 0,Y 509.891,Z 66.473,A -85,B 0,C 180,E1 -5282.055,E2 -5282.055} C_VEL
LIN {X 0,Y 509.874,Z 66.47,A -85,B 0,C 180,E1 -5284.704,E2 -5284.704} C_VEL
LIN {X 0,Y 509.833,Z 66.48,A -85,B 0,C 180,E1 -5287.455,E2 -5287.455} C_VEL
LIN {X 0,Y 509.914,Z 66.471,A -85,B 0,C 180,E1 -5289.845,E2 -5289.845} C_VEL
LIN {X 0,Y 509.882,Z 66.473,A -85,B 0,C 180,E1 -5293.175,E2 -5293.175} C_VEL
LIN {X 0,Y 509.871,Z 66.477,A -85,B 0,C 180,E1 -5295.634,E2 -5295.634} C_VEL
LIN {X 0,Y 509.91,Z 66.469,A -85,B 0,C 180,E1 -5298.874,E2 -5298.874} C_VEL
LIN {X 0,Y 509.949,Z 66.462,A -85,B 0,C 180,E1 -5302.078,E2 -5302.078} C_VEL
LIN {X 0,Y 509.983,Z 66.458,A -85,B 0,C 180,E1 -5304.464,E2 -5304.464} C_VEL
LIN {X 0,Y 510.053,Z 66.45,A -85,B 0,C 180,E1 -5307.631,E2 -5307.631} C_VEL
LIN {X 0,Y 510.061,Z 66.453,A -85,B 0,C 180,E1 -5310.789,E2 -5310.789} C_VEL
LIN {X 0,Y 509.952,Z 66.466,A -85,B 0,C 180,E1 -5313.16,E2 -5313.16} C_VEL
LIN {X 0,Y 509.98,Z 66.46,A -85,B 0,C 180,E1 -5316.33,E2 -5316.33} C_VEL
LIN {X 0,Y 509.913,Z 66.472,A -85,B 0,C 180,E1 -5318.72,E2 -5318.72} C_VEL
LIN {X 0,Y 509.901,Z 66.468,A -85,B 0,C 180,E1 -5321.932,E2 -5321.932} C_VEL
LIN {X 0,Y 509.89,Z 66.469,A -85,B 0,C 180,E1 -5325.242,E2 -5325.242} C_VEL
LIN {X 0,Y 509.885,Z 66.472,A -85,B 0,C 180,E1 -5328.001,E2 -5328.001} C_VEL
LIN {X 0,Y 509.847,Z 66.475,A -85,B 0,C 180,E1 -5331.002,E2 -5331.002} C_VEL
LIN {X 0,Y 509.834,Z 66.476,A -85,B 0,C 180,E1 -5333.563,E2 -5333.563} C_VEL
LIN {X 0,Y 509.909,Z 66.471,A -85,B 0,C 180,E1 -5336.379,E2 -5336.379} C_VEL
LIN {X 0,Y 509.874,Z 66.464,A -85,B 0,C 180,E1 -5338.844,E2 -5338.844} C_VEL
LIN {X 0,Y 509.823,Z 66.479,A -85,B 0,C 180,E1 -5341.59,E2 -5341.59} C_VEL
LIN {X 0,Y 509.851,Z 66.46,A -85,B 0,C 180,E1 -5344.413,E2 -5344.413} C_VEL
LIN {X 0,Y 509.816,Z 66.478,A -85,B 0,C 180,E1 -5347.341,E2 -5347.341} C_VEL
LIN {X 0,Y 509.835,Z 66.467,A -85,B 0,C 180,E1 -5350.382,E2 -5350.382} C_VEL
LIN {X 0,Y 509.816,Z 66.464,A -85,B 0,C 180,E1 -5353.062,E2 -5353.062} C_VEL
LIN {X 0,Y 509.828,Z 66.479,A -85,B 0,C 180,E1 -5355.793,E2 -5355.793} C_VEL
LIN {X 0,Y 509.862,Z 66.468,A -85,B 0,C 180,E1 -5358.576,E2 -5358.576} C_VEL
LIN {X 0,Y 509.849,Z 66.475,A -85,B 0,C 180,E1 -5361.787,E2 -5361.787} C_VEL
LIN {X 0,Y 509.844,Z 66.472,A -85,B 0,C 180,E1 -5364.624,E2 -5364.624} C_VEL
LIN {X 0,Y 509.861,Z 66.474,A -85,B 0,C 180,E1 -5367.481,E2 -5367.481} C_VEL
LIN {X 0,Y 509.856,Z 66.471,A -85,B 0,C 180,E1 -5370.274,E2 -5370.274} C_VEL
LIN {X 0,Y 509.883,Z 66.466,A -85,B 0,C 180,E1 -5372.945,E2 -5372.945} C_VEL
LIN {X 0,Y 509.868,Z 66.47,A -85,B 0,C 180,E1 -5375.574,E2 -5375.574} C_VEL
LIN {X 0,Y 509.849,Z 66.471,A -85,B 0,C 180,E1 -5378.999,E2 -5378.999} C_VEL
LIN {X 0,Y 509.887,Z 66.46,A -85,B 0,C 180,E1 -5382,E2 -5382} C_VEL
LIN {X 0,Y 509.909,Z 66.469,A -85,B 0,C 180,E1 -5384.819,E2 -5384.819} C_VEL
LIN {X 0,Y 509.943,Z 66.462,A -85,B 0,C 180,E1 -5388.101,E2 -5388.101} C_VEL
LIN {X 0,Y 509.914,Z 66.456,A -85,B 0,C 180,E1 -5391.28,E2 -5391.28} C_VEL
LIN {X 0,Y 509.978,Z 66.455,A -85,B 0,C 180,E1 -5393.671,E2 -5393.671} C_VEL
LIN {X 0,Y 510.055,Z 66.446,A -85,B 0,C 180,E1 -5397.631,E2 -5397.631} C_VEL
LIN {X 0,Y 510.064,Z 66.437,A -85,B 0,C 180,E1 -5400.79,E2 -5400.79} C_VEL
LIN {X 0,Y 509.953,Z 66.457,A -85,B 0,C 180,E1 -5403.161,E2 -5403.161} C_VEL
LIN {X 0,Y 509.979,Z 66.455,A -85,B 0,C 180,E1 -5406.33,E2 -5406.33} C_VEL
LIN {X 0,Y 509.915,Z 66.455,A -85,B 0,C 180,E1 -5408.721,E2 -5408.721} C_VEL
LIN {X 0,Y 509.905,Z 66.467,A -85,B 0,C 180,E1 -5411.932,E2 -5411.932} C_VEL
LIN {X 0,Y 509.895,Z 66.469,A -85,B 0,C 180,E1 -5415.242,E2 -5415.242} C_VEL
LIN {X 0,Y 509.883,Z 66.459,A -85,B 0,C 180,E1 -5417.999,E2 -5417.999} C_VEL
LIN {X 0,Y 509.852,Z 66.47,A -85,B 0,C 180,E1 -5421.002,E2 -5421.002} C_VEL
LIN {X 0,Y 509.871,Z 66.468,A -85,B 0,C 180,E1 -5424.426,E2 -5424.426} C_VEL
LIN {X 0,Y 509.885,Z 66.466,A -85,B 0,C 180,E1 -5427.056,E2 -5427.056} C_VEL
LIN {X 0,Y 509.858,Z 66.471,A -85,B 0,C 180,E1 -5429.751,E2 -5429.751} C_VEL
LIN {X 0,Y 509.874,Z 66.474,A -85,B 0,C 180,E1 -5432.774,E2 -5432.774} C_VEL
LIN {X 0,Y 509.83,Z 66.473,A -85,B 0,C 180,E1 -5435.579,E2 -5435.579} C_VEL
LIN {X 0,Y 509.852,Z 66.474,A -85,B 0,C 180,E1 -5438.338,E2 -5438.338} C_VEL
LIN {X 0,Y 509.857,Z 66.471,A -85,B 0,C 180,E1 -5441.426,E2 -5441.426} C_VEL
LIN {X 0,Y 509.84,Z 66.477,A -85,B 0,C 180,E1 -5444.67,E2 -5444.67} C_VEL
LIN {X 0,Y 509.834,Z 66.473,A -85,B 0,C 180,E1 -5447.51,E2 -5447.51} C_VEL
LIN {X 0,Y 509.847,Z 66.473,A -85,B 0,C 180,E1 -5450.648,E2 -5450.648} C_VEL
LIN {X 0,Y 509.836,Z 66.475,A -85,B 0,C 180,E1 -5453.648,E2 -5453.648} C_VEL
LIN {X 0,Y 509.863,Z 66.474,A -85,B 0,C 180,E1 -5456.54,E2 -5456.54} C_VEL
LIN {X 0,Y 509.848,Z 66.475,A -85,B 0,C 180,E1 -5459.335,E2 -5459.335} C_VEL
LIN {X 0,Y 509.897,Z 66.471,A -85,B 0,C 180,E1 -5462.055,E2 -5462.055} C_VEL
LIN {X 0,Y 509.954,Z 66.684,A -85,B 0,C 180,E1 -5463.704,E2 -5463.704} C_VEL
LIN {X 0,Y 511.145,Z 74.323,A -85,B 0,C 180,E1 -5465.406,E2 -5465.406} C_VEL
LIN {X 0,Y 510.764,Z 87.798,A -85,B 0,C 180,E1 -5468.191,E2 -5468.191} C_VEL
LIN {X 0,Y 510.388,Z 101.328,A -85,B 0,C 180,E1 -5470.911,E2 -5470.911} C_VEL
LIN {X 0,Y 510.136,Z 114.75,A -85,B 0,C 180,E1 -5473.595,E2 -5473.595} C_VEL
LIN {X 0,Y 509.977,Z 118.814,A -85,B 0,C 180,E1 -5474.397,E2 -5474.397} C_VEL
LIN {X 0,Y 511.059,Z 125.674,A -85,B 0,C 180,E1 -5474.561,E2 -5474.561} C_VEL
LIN {X 0,Y 512.181,Z 132.395,A -85,B 0,C 180,E1 -5474.691,E2 -5474.691} C_VEL
LIN {X 0,Y 511.752,Z 223.667,A -85,B 0,C 180,E1 -5475.993,E2 -5475.993} C_VEL
LIN {X 0,Y 511.519,Z 234.437,A -85,B 0,C 180,E1 -5476.24,E2 -5476.24} C_VEL
LIN {X 0,Y 511.361,Z 243.542,A -85,B 0,C 180,E1 -5476.539,E2 -5476.539} C_VEL
LIN {X 0,Y 511.106,Z 252.9,A -85,B 0,C 180,E1 -5476.937,E2 -5476.937} C_VEL
LIN {X 0,Y 510.851,Z 262.531,A -85,B 0,C 180,E1 -5477.454,E2 -5477.454} C_VEL
LIN {X 0,Y 510.545,Z 272.044,A -85,B 0,C 180,E1 -5478.084,E2 -5478.084} C_VEL
LIN {X 0,Y 510.304,Z 280.776,A -85,B 0,C 180,E1 -5478.783,E2 -5478.783} C_VEL
LIN {X 0,Y 510.064,Z 288.173,A -85,B 0,C 180,E1 -5479.481,E2 -5479.481} C_VEL
LIN {X 0,Y 509.881,Z 295.395,A -85,B 0,C 180,E1 -5480.279,E2 -5480.279} C_VEL
LIN {X 0,Y 509.649,Z 301.596,A -85,B 0,C 180,E1 -5481.075,E2 -5481.075} C_VEL
LIN {X 0,Y 509.489,Z 308.133,A -85,B 0,C 180,E1 -5482.071,E2 -5482.071} C_VEL
LIN {X 0,Y 509.332,Z 313.686,A -85,B 0,C 180,E1 -5483.085,E2 -5483.085} C_VEL
LIN {X 0,Y 509.289,Z 318.122,A -85,B 0,C 180,E1 -5484.059,E2 -5484.059} C_VEL
LIN {X 0,Y 509.188,Z 322.441,A -85,B 0,C 180,E1 -5485.25,E2 -5485.25} C_VEL
LIN {X 0,Y 509.245,Z 324.807,A -85,B 0,C 180,E1 -5486.043,E2 -5486.043} C_VEL
LIN {X 0,Y 509.201,Z 326.601,A -85,B 0,C 180,E1 -5486.835,E2 -5486.835} C_VEL
LIN {X 0,Y 509.113,Z 329.039,A -85,B 0,C 180,E1 -5488.418,E2 -5488.418} C_VEL
LIN {X 0,Y 509.077,Z 329.625,A -85,B 0,C 180,E1 -5489.209,E2 -5489.209} C_VEL
LIN {X 0,Y 509.077,Z 329.625,A -85,B 0,C 180,E1 -5490.791,E2 -5490.791} C_VEL
LIN {X 0,Y 509.113,Z 329.039,A -85,B 0,C 180,E1 -5491.582,E2 -5491.582} C_VEL
LIN {X 0,Y 509.201,Z 326.601,A -85,B 0,C 180,E1 -5493.165,E2 -5493.165} C_VEL
LIN {X 0,Y 509.205,Z 323.657,A -85,B 0,C 180,E1 -5494.354,E2 -5494.354} C_VEL
LIN {X 0,Y 509.279,Z 319.675,A -85,B 0,C 180,E1 -5495.543,E2 -5495.543} C_VEL
LIN {X 0,Y 509.304,Z 314.739,A -85,B 0,C 180,E1 -5496.696,E2 -5496.696} C_VEL
LIN {X 0,Y 509.457,Z 309.288,A -85,B 0,C 180,E1 -5497.73,E2 -5497.73} C_VEL
LIN {X 0,Y 509.635,Z 302.973,A -85,B 0,C 180,E1 -5498.725,E2 -5498.725} C_VEL
LIN {X 0,Y 509.82,Z 297.021,A -85,B 0,C 180,E1 -5499.522,E2 -5499.522} C_VEL
